# B&R Automation Studio project NAELD004C00R10L518F00 (part 11)

#### Act_OptP0921RstMnl.st
```iecst
ACTION Act_OptP0921RstMnl:

	IF EDGEPOS((bManualMod = FALSE) OR (p_eInShutterStatus = Error) OR (p_eInShutterStatus2 = Error) OR (p_eInShutterStatus3 = Error)) THEN

		eInShutterAct	:= PneuActIdle;
		eInShutterAct2	:= PneuActIdle;
		eInShutterAct3	:= PneuActIdle;

		tyP0921InletNOutletShutter.tyInletShutterDC.tyBtnClose.bRtCompl	:= FALSE;
		tyP0921InletNOutletShutter.tyInletShutterDC.tyBtnClose.bValue	:= FALSE;
		tyP0921InletNOutletShutter.tyInletShutterDC.tyBtnOpen.bRtCompl	:= FALSE;
		tyP0921InletNOutletShutter.tyInletShutterDC.tyBtnOpen.bValue	:= TRUE;

		tyP0921InletNOutletShutter.tyInletShutterFB.tyBtnClose.bRtCompl	:= FALSE;
		tyP0921InletNOutletShutter.tyInletShutterFB.tyBtnClose.bValue	:= FALSE;
		tyP0921InletNOutletShutter.tyInletShutterFB.tyBtnOpen.bRtCompl	:= FALSE;
		tyP0921InletNOutletShutter.tyInletShutterFB.tyBtnOpen.bValue	:= FALSE;

		//in shutt 2
		tyP0921InletNOutletShutter.tyInletShutterDC2.tyBtnClose.bRtCompl	:= FALSE;
		tyP0921InletNOutletShutter.tyInletShutterDC2.tyBtnClose.bValue	:= FALSE;
		tyP0921InletNOutletShutter.tyInletShutterDC2.tyBtnOpen.bRtCompl	:= FALSE;
		tyP0921InletNOutletShutter.tyInletShutterDC2.tyBtnOpen.bValue	:= TRUE;

		tyP0921InletNOutletShutter.tyInletShutterFB2.tyBtnClose.bRtCompl	:= FALSE;
		tyP0921InletNOutletShutter.tyInletShutterFB2.tyBtnClose.bValue	:= FALSE;
		tyP0921InletNOutletShutter.tyInletShutterFB2.tyBtnOpen.bRtCompl	:= FALSE;
		tyP0921InletNOutletShutter.tyInletShutterFB2.tyBtnOpen.bValue	:= FALSE;

		//in shutt3
		tyP0921InletNOutletShutter.tyInletShutterDC3.tyBtnClose.bRtCompl	:= FALSE;
		tyP0921InletNOutletShutter.tyInletShutterDC3.tyBtnClose.bValue	:= FALSE;
		tyP0921InletNOutletShutter.tyInletShutterDC3.tyBtnOpen.bRtCompl	:= FALSE;
		tyP0921InletNOutletShutter.tyInletShutterDC3.tyBtnOpen.bValue	:= TRUE;

		tyP0921InletNOutletShutter.tyInletShutterFB3.tyBtnClose.bRtCompl	:= FALSE;
		tyP0921InletNOutletShutter.tyInletShutterFB3.tyBtnClose.bValue	:= FALSE;
		tyP0921InletNOutletShutter.tyInletShutterFB3.tyBtnOpen.bRtCompl	:= FALSE;
		tyP0921InletNOutletShutter.tyInletShutterFB3.tyBtnOpen.bValue	:= FALSE;

	END_IF

	IF EDGEPOS((bManualMod = FALSE) OR (p_eOutShutterStatus = Error) OR (p_eOutShutterStatus2 = Error) ) THEN

		eOutShutterAct	:= PneuActIdle;
		eOutShutterAct2	:= PneuActIdle;

		tyP0921InletNOutletShutter.tyOutletShutterDC.tyBtnClose.bRtCompl	:= FALSE;
		tyP0921InletNOutletShutter.tyOutletShutterDC.tyBtnClose.bValue		:= FALSE;
		tyP0921InletNOutletShutter.tyOutletShutterDC.tyBtnOpen.bRtCompl		:= FALSE;
		tyP0921InletNOutletShutter.tyOutletShutterDC.tyBtnOpen.bValue		:= FALSE;

		tyP0921InletNOutletShutter.tyOutletShutterFB.tyBtnClose.bRtCompl	:= FALSE;
		tyP0921InletNOutletShutter.tyOutletShutterFB.tyBtnClose.bValue		:= FALSE;
		tyP0921InletNOutletShutter.tyOutletShutterFB.tyBtnOpen.bRtCompl		:= FALSE;
		tyP0921InletNOutletShutter.tyOutletShutterFB.tyBtnOpen.bValue		:= FALSE;

		tyP0921InletNOutletShutter.tyOutletShutterDC2.tyBtnClose.bRtCompl	:= FALSE;
		tyP0921InletNOutletShutter.tyOutletShutterDC2.tyBtnClose.bValue		:= FALSE;
		tyP0921InletNOutletShutter.tyOutletShutterDC2.tyBtnOpen.bRtCompl	:= FALSE;
		tyP0921InletNOutletShutter.tyOutletShutterDC2.tyBtnOpen.bValue		:= FALSE;

		tyP0921InletNOutletShutter.tyOutletShutterFB2.tyBtnClose.bRtCompl	:= FALSE;
		tyP0921InletNOutletShutter.tyOutletShutterFB2.tyBtnClose.bValue		:= FALSE;
		tyP0921InletNOutletShutter.tyOutletShutterFB2.tyBtnOpen.bRtCompl	:= FALSE;
		tyP0921InletNOutletShutter.tyOutletShutterFB2.tyBtnOpen.bValue		:= FALSE;

	END_IF

	IF EDGEPOS(bManualMod = FALSE) THEN

		//In Shutter
		tyP0921InletNOutletShutter.tyInletShutterCom.tyBtnSwitch.bValue		:= FALSE;
		tyP0921InletNOutletShutter.tyInletShutterCom2.tyBtnSwitch.bValue		:= FALSE;

		fUIInRtStatHide(ADR(tyP0921InletNOutletShutter.tyInletShutterDC.tyLyr.uiRtStat));
		fUIInRtStatOff(ADR(tyP0921InletNOutletShutter.tyInletShutterFB.tyLyr.uiRtStat));

		//Out Shutter
		tyP0921InletNOutletShutter.tyOutletShutterCom.tyBtnSwitch.bValue   := FALSE;
		tyP0921InletNOutletShutter.tyOutletShutterCom2.tyBtnSwitch.bValue   := FALSE;

		fUIInRtStatHide(ADR(tyP0921InletNOutletShutter.tyOutletShutterDC.tyLyr.uiRtStat));
		fUIInRtStatOff(ADR(tyP0921InletNOutletShutter.tyOutletShutterFB.tyLyr.uiRtStat));

	END_IF

END_ACTION
```

#### Act_OptP0921InletShutterChgLyr2.st
```iecst
ACTION Act_OptP0921InletShutterChgLyr2:

//	tyP0921InletNOutletShutter.tyInletShutterFB.tyLyr.uiRtStat.0	:= NOT(p_tyNtParamCurr.bProjInletShutPrep);

	IF p_tyNtParamCurr.bProjInletShutPrep THEN
		IF tyP0921InletNOutletShutter.tyInletShutterCom2.tyBtnSwitch.bRtCompl THEN
			tyP0921InletNOutletShutter.tyInletShutterCom2.tyBtnSwitch.bRtCompl := FALSE;

			IF tyP0921InletNOutletShutter.tyInletShutterCom2.tyBtnSwitch.bValue = TRUE THEN
				fUIInRtStatOff(ADR(tyP0921InletNOutletShutter.tyInletShutterDC2.tyLyr.uiRtStat));
				fUIInRtStatHide(ADR(tyP0921InletNOutletShutter.tyInletShutterFB2.tyLyr.uiRtStat));
			ELSE
				fUIInRtStatHide(ADR(tyP0921InletNOutletShutter.tyInletShutterDC2.tyLyr.uiRtStat));
				fUIInRtStatOff(ADR(tyP0921InletNOutletShutter.tyInletShutterFB2.tyLyr.uiRtStat));
			END_IF

		END_IF
	ELSE
		fUIInRtStatHide(ADR(tyP0921InletNOutletShutter.tyInletShutterDC2.tyLyr.uiRtStat));
		fUIInRtStatHide(ADR(tyP0921InletNOutletShutter.tyInletShutterFB2.tyLyr.uiRtStat));

	END_IF

END_ACTION
```

#### Act_OptP0921InletShutterSen2.st
```iecst
ACTION Act_OptP0921InletShutterSen2:

	tyP0921InletNOutletShutter.tyInletShutterCom2.tyBtnOpenRS.bValue		:= p_tyDI.bInShutterOpenRS2;
	tyP0921InletNOutletShutter.tyInletShutterCom2.tyBtnCloseRS.bValue	:= p_tyDI.bInShutterCloseRS2;

	//Machine Bitmap ,13close 14open
	IF   (p_tyNtParamCurr.eProjMag = LDMagDual AND p_tyNtParamCurr.bMagAutoVerifyPrep = FALSE)
		OR (p_tyNtParamCurr.eProjMag = LDMagTriple AND p_tyNtParamCurr.bMagAutoVerifyPrep = FALSE)
		OR (p_tyNtParamCurr.eProjMag = LDMagDual AND p_tyNtParamCurr.bMagAutoVerifyPrep = TRUE)
		THEN
		IF p_tyDI.bInShutterOpenRS2 = TRUE THEN
			tyP0921InletNOutletShutter.tyInletShutterCom2.tyBitmapMc.uiValueIdx	:= 2;
		ELSIF p_tyNtParamCurr.bProjCurtainSenPrep THEN
			tyP0921InletNOutletShutter.tyInletShutterCom2.tyBitmapMc.uiValueIdx	:= 0+4; //16
		ELSE
			tyP0921InletNOutletShutter.tyInletShutterCom2.tyBitmapMc.uiValueIdx	:= 0;
		END_IF
	ELSIF p_tyNtParamCurr.eProjMag = LDMagTriple AND p_tyNtParamCurr.bMagAutoVerifyPrep = TRUE
		THEN
		IF p_tyDI.bInShutterOpenRS2 = TRUE THEN
			tyP0921InletNOutletShutter.tyInletShutterCom2.tyBitmapMc.uiValueIdx	:= 28;
		ELSE
			tyP0921InletNOutletShutter.tyInletShutterCom2.tyBitmapMc.uiValueIdx	:= 27;
		END_IF

	ELSIF p_tyNtParamCurr.eProjMag = LDMagQuadruple AND p_tyNtParamCurr.bMagAutoVerifyPrep = TRUE
		THEN
		IF p_tyDI.bInShutterOpenRS2 = TRUE THEN
			tyP0921InletNOutletShutter.tyInletShutterCom2.tyBitmapMc.uiValueIdx	:= 51;
		ELSE
			tyP0921InletNOutletShutter.tyInletShutterCom2.tyBitmapMc.uiValueIdx	:= 50;
		END_IF
	END_IF

	IF p_tyNtParamCurr.eProjMag = LDMagTriple AND p_tyNtParamCurr.bProjLifterMagPlatform THEN
		IF 	tyP0921InletNOutletShutter.tyInletShutterCom2.tyBitmapMc.uiValueIdx < 400 THEN
			tyP0921InletNOutletShutter.tyInletShutterCom2.tyBitmapMc.uiValueIdx	:= tyP0921InletNOutletShutter.tyInletShutterCom2.tyBitmapMc.uiValueIdx + 400;
		END_IF
	ELSIF p_tyNtParamCurr.eProjMag = LDMagTriple AND p_tyNtParamCurr.bMagAutoVerifyPrep = FALSE AND p_tyNtParamCurr.bProjMotorizedPullerPrep = FALSE
		THEN
		IF 	tyP0921InletNOutletShutter.tyInletShutterCom2.tyBitmapMc.uiValueIdx < 100 THEN
			tyP0921InletNOutletShutter.tyInletShutterCom2.tyBitmapMc.uiValueIdx	:= tyP0921InletNOutletShutter.tyInletShutterCom2.tyBitmapMc.uiValueIdx + 100;
		END_IF
	ELSIF p_tyNtParamCurr.eProjMag = LDMagTriple AND p_tyNtParamCurr.bMagAutoVerifyPrep = FALSE AND p_tyNtParamCurr.bProjMotorizedPullerPrep
		AND p_tyNtParamCurr.bProjCurtainSenPrep THEN //curtain
		IF 	tyP0921InletNOutletShutter.tyInletShutterCom2.tyBitmapMc.uiValueIdx < 375-13-1 THEN
			tyP0921InletNOutletShutter.tyInletShutterCom2.tyBitmapMc.uiValueIdx	:= tyP0921InletNOutletShutter.tyInletShutterCom2.tyBitmapMc.uiValueIdx + 375-13-1;
		END_IF
	ELSIF (p_tyNtParamCurr.eProjMag = LDMagDual OR p_tyNtParamCurr.eProjMag = LDMagTriple)
		AND p_tyNtParamCurr.bMagAutoVerifyPrep = TRUE
		THEN
		IF 	tyP0921InletNOutletShutter.tyInletShutterCom2.tyBitmapMc.uiValueIdx < 200 THEN
			tyP0921InletNOutletShutter.tyInletShutterCom2.tyBitmapMc.uiValueIdx	:= tyP0921InletNOutletShutter.tyInletShutterCom2.tyBitmapMc.uiValueIdx + 200;
		END_IF
	ELSIF (p_tyNtParamCurr.eProjMag = LDMagDual OR p_tyNtParamCurr.eProjMag = LDMagTriple) AND p_tyNtParamCurr.bMagAutoVerifyPrep = FALSE AND  p_tyNtParamCurr.bProjMotorizedPullerPrep = FALSE THEN
		IF 	tyP0921InletNOutletShutter.tyInletShutterCom2.tyBitmapMc.uiValueIdx < 200 THEN
			IF p_tyNtParamCurr.bProjLifterMagPlatform THEN
				tyP0921InletNOutletShutter.tyInletShutterCom2.tyBitmapMc.uiValueIdx	:= tyP0921InletNOutletShutter.tyInletShutterCom2.tyBitmapMc.uiValueIdx + 247;
			ELSE
				tyP0921InletNOutletShutter.tyInletShutterCom2.tyBitmapMc.uiValueIdx	:= tyP0921InletNOutletShutter.tyInletShutterCom2.tyBitmapMc.uiValueIdx + 200;
			END_IF
		END_IF
	ELSIF (p_tyNtParamCurr.eProjMag = LDMagDual OR p_tyNtParamCurr.eProjMag = LDMagTriple) AND p_tyNtParamCurr.bMagAutoVerifyPrep = FALSE AND p_tyNtParamCurr.bProjMotorizedPullerPrep = TRUE
		THEN
		IF 	tyP0921InletNOutletShutter.tyInletShutterCom2.tyBitmapMc.uiValueIdx < 300 THEN
			tyP0921InletNOutletShutter.tyInletShutterCom2.tyBitmapMc.uiValueIdx	:= tyP0921InletNOutletShutter.tyInletShutterCom2.tyBitmapMc.uiValueIdx + 300;
		END_IF
	END_IF
END_ACTION
```

#### Act_OptP0921InletShutterFB2.st
```iecst
ACTION Act_OptP0921InletShutterFB2:

	IF tyP0921InletNOutletShutter.tyInletShutterCom2.tyBtnSwitch.bValue = FALSE THEN

		IF tyP0921InletNOutletShutter.tyInletShutterFB2.tyBtnOpen.bRtCompl = TRUE THEN
			tyP0921InletNOutletShutter.tyInletShutterFB2.tyBtnOpen.bRtCompl	:= FALSE;

			tyP0921InletNOutletShutter.tyInletShutterFB2.tyBtnOpen.bValue	:= TRUE;
			tyP0921InletNOutletShutter.tyInletShutterFB2.tyBtnClose.bValue	:= FALSE;

		ELSIF tyP0921InletNOutletShutter.tyInletShutterFB2.tyBtnClose.bRtCompl = TRUE THEN
			tyP0921InletNOutletShutter.tyInletShutterFB2.tyBtnClose.bRtCompl	:= FALSE;

			tyP0921InletNOutletShutter.tyInletShutterFB2.tyBtnClose.bValue	:= TRUE;
			tyP0921InletNOutletShutter.tyInletShutterFB2.tyBtnOpen.bValue	:= FALSE;
		END_IF

		IF tyP0921InletNOutletShutter.tyInletShutterFB2.tyBtnOpen.bValue = TRUE THEN
			eInShutterAct2	:= PneuActRet;

			IF p_eInShutterStat2 = PneuActRet AND p_eInShutterStatus2 = Done THEN
				eInShutterAct2	:= PneuActIdle;

				tyP0921InletNOutletShutter.tyInletShutterFB2.tyBtnOpen.bValue	:= FALSE;
			ELSIF p_eInShutterStatus2 = Error THEN
				tyP0921InletNOutletShutter.tyInletShutterFB2.tyBtnOpen.bValue	:= FALSE;
			END_IF

		ELSIF tyP0921InletNOutletShutter.tyInletShutterFB2.tyBtnClose.bValue = TRUE THEN
			eInShutterAct2	:= PneuActExt;

			IF p_eInShutterStat2 = PneuActExt AND p_eInShutterStatus2 = Done THEN
				eInShutterAct2	:= PneuActIdle;

				tyP0921InletNOutletShutter.tyInletShutterFB2.tyBtnClose.bValue := FALSE;
			ELSIF p_eInShutterStatus2 = Error THEN
				tyP0921InletNOutletShutter.tyInletShutterFB2.tyBtnClose.bValue := FALSE;
			END_IF
		END_IF

		//Update Direct Control Status
		tyP0921InletNOutletShutter.tyInletShutterDC2.tyBtnOpen.bRtCompl	:= FALSE;
		tyP0921InletNOutletShutter.tyInletShutterDC2.tyBtnClose.bRtCompl	:= FALSE;
		tyP0921InletNOutletShutter.tyInletShutterDC2.tyBtnOpen.bValue	:= p_bInShutterRetCtrl2;
		tyP0921InletNOutletShutter.tyInletShutterDC2.tyBtnClose.bValue	:= p_bInShutterExtCtrl2;

	END_IF

END_ACTION
```

#### Act_OptP0921InletShutterFBStat2.st
```iecst
ACTION Act_OptP0921InletShutterFBStat2:

	tyP0921InletNOutletShutter.tyInletShutterFB2.tyStringStat.sValue	:= p_sInShutterStatTxt2;

END_ACTION
```

#### Act_OptP0921InletShutterDC2.st
```iecst
ACTION Act_OptP0921InletShutterDC2:

	IF tyP0921InletNOutletShutter.tyInletShutterCom2.tyBtnSwitch.bValue = TRUE THEN
		IF p_bInShutterTwoCtrlOut2 = FALSE THEN
			IF tyP0921InletNOutletShutter.tyInletShutterDC2.tyBtnOpen.bRtCompl = TRUE THEN
				tyP0921InletNOutletShutter.tyInletShutterDC2.tyBtnOpen.bValue	:= TRUE;
				tyP0921InletNOutletShutter.tyInletShutterDC2.tyBtnClose.bValue	:= FALSE;

				eInShutterAct2	:= PneuActSetRet;

				IF p_eInShutterStat2 = PneuActSetRet AND p_eInShutterStatus2 = Done THEN
					eInShutterAct2	:= PneuActIdle;

					tyP0921InletNOutletShutter.tyInletShutterDC2.tyBtnOpen.bRtCompl	:= FALSE;
				END_IF

			ELSIF tyP0921InletNOutletShutter.tyInletShutterDC2.tyBtnClose.bRtCompl = TRUE THEN
				tyP0921InletNOutletShutter.tyInletShutterDC2.tyBtnClose.bValue	:= TRUE;
				tyP0921InletNOutletShutter.tyInletShutterDC2.tyBtnOpen.bValue	:= FALSE;

				eInShutterAct2	:= PneuActSetExt;

				IF p_eInShutterStat2 = PneuActSetExt AND p_eInShutterStatus2 = Done THEN
					eInShutterAct2	:= PneuActIdle;

					tyP0921InletNOutletShutter.tyInletShutterDC2.tyBtnClose.bRtCompl	:= FALSE;
				END_IF
			END_IF

		ELSE
			IF (tyP0921InletNOutletShutter.tyInletShutterDC2.tyBtnOpen.bRtCompl = TRUE) OR (tyP0921InletNOutletShutter.tyInletShutterDC2.tyBtnClose.bRtCompl = TRUE) THEN
				IF (tyP0921InletNOutletShutter.tyInletShutterDC2.tyBtnOpen.bValue = TRUE) AND (tyP0921InletNOutletShutter.tyInletShutterDC2.tyBtnClose.bValue = TRUE) THEN
					eInShutterAct2	:= PneuActSetAll;

					IF p_eInShutterStat2 = PneuActSetAll AND p_eInShutterStatus2 = Done THEN
						eInShutterAct2	:= PneuActIdle;

						tyP0921InletNOutletShutter.tyInletShutterDC2.tyBtnOpen.bRtCompl	:= FALSE;
						tyP0921InletNOutletShutter.tyInletShutterDC2.tyBtnClose.bRtCompl	:= FALSE;
					END_IF

				ELSIF (tyP0921InletNOutletShutter.tyInletShutterDC2.tyBtnOpen.bValue = TRUE) AND (tyP0921InletNOutletShutter.tyInletShutterDC2.tyBtnClose.bValue = FALSE) THEN
					eInShutterAct2	:= PneuActSetRet;

					IF p_eInShutterStat2 = PneuActSetRet AND p_eInShutterStatus2 = Done THEN
						eInShutterAct2	:= PneuActIdle;

						tyP0921InletNOutletShutter.tyInletShutterDC2.tyBtnOpen.bRtCompl	:= FALSE;
						tyP0921InletNOutletShutter.tyInletShutterDC2.tyBtnClose.bRtCompl	:= FALSE;
					END_IF

				ELSIF (tyP0921InletNOutletShutter.tyInletShutterDC2.tyBtnOpen.bValue = FALSE) AND (tyP0921InletNOutletShutter.tyInletShutterDC2.tyBtnClose.bValue = TRUE) THEN
					eInShutterAct2	:= PneuActSetExt;

					IF p_eInShutterStat2 = PneuActSetExt AND p_eInShutterStatus2 = Done THEN
						eInShutterAct2	:= PneuActIdle;

						tyP0921InletNOutletShutter.tyInletShutterDC2.tyBtnOpen.bRtCompl	:= FALSE;
						tyP0921InletNOutletShutter.tyInletShutterDC2.tyBtnClose.bRtCompl	:= FALSE;
					END_IF

				ELSE
					eInShutterAct2	:= PneuActRstAll;

					IF p_eInShutterStat2 = PneuActRstAll AND p_eInShutterStatus2 = Done THEN
						eInShutterAct2	:= PneuActIdle;

						tyP0921InletNOutletShutter.tyInletShutterDC2.tyBtnOpen.bRtCompl	:= FALSE;
						tyP0921InletNOutletShutter.tyInletShutterDC2.tyBtnClose.bRtCompl	:= FALSE;
					END_IF

				END_IF
			END_IF
		END_IF

		tyP0921InletNOutletShutter.tyInletShutterFB2.tyBtnClose.bRtCompl	:= FALSE;
		tyP0921InletNOutletShutter.tyInletShutterFB2.tyBtnClose.bValue	:= FALSE;
		tyP0921InletNOutletShutter.tyInletShutterFB2.tyBtnOpen.bRtCompl	:= FALSE;
		tyP0921InletNOutletShutter.tyInletShutterFB2.tyBtnOpen.bValue	:= FALSE;

	END_IF

END_ACTION
```

#### Act_OptP0921InletShutterChgLyr3.st
```iecst
ACTION Act_OptP0921InletShutterChgLyr3:

//	tyP0921InletNOutletShutter.tyInletShutterFB2.tyLyr.uiRtStat.0	:= NOT(p_tyNtParamCurr.bProjInletShutPrep);

	IF p_tyNtParamCurr.bProjInletShutPrep THEN
		IF tyP0921InletNOutletShutter.tyInletShutterCom3.tyBtnSwitch.bRtCompl THEN
			tyP0921InletNOutletShutter.tyInletShutterCom3.tyBtnSwitch.bRtCompl := FALSE;

			IF tyP0921InletNOutletShutter.tyInletShutterCom3.tyBtnSwitch.bValue = TRUE THEN
				fUIInRtStatOff(ADR(tyP0921InletNOutletShutter.tyInletShutterDC3.tyLyr.uiRtStat));
				fUIInRtStatHide(ADR(tyP0921InletNOutletShutter.tyInletShutterFB3.tyLyr.uiRtStat));
			ELSE
				fUIInRtStatHide(ADR(tyP0921InletNOutletShutter.tyInletShutterDC3.tyLyr.uiRtStat));
				fUIInRtStatOff(ADR(tyP0921InletNOutletShutter.tyInletShutterFB3.tyLyr.uiRtStat));
			END_IF

		END_IF
	ELSE
		fUIInRtStatHide(ADR(tyP0921InletNOutletShutter.tyInletShutterDC3.tyLyr.uiRtStat));
		fUIInRtStatHide(ADR(tyP0921InletNOutletShutter.tyInletShutterFB3.tyLyr.uiRtStat));

	END_IF

END_ACTION
```

#### Act_OptP0921InletShutterSen3.st
```iecst
ACTION Act_OptP0921InletShutterSen3:

	tyP0921InletNOutletShutter.tyInletShutterCom3.tyBtnOpenRS.bValue		:= p_tyDI.bInShutterOpenRS3;
	tyP0921InletNOutletShutter.tyInletShutterCom3.tyBtnCloseRS.bValue	:= p_tyDI.bInShutterCloseRS3;

	//Machine Bitmap, 15close ,16open
	IF   (p_tyNtParamCurr.eProjMag = LDMagDual AND p_tyNtParamCurr.bMagAutoVerifyPrep = FALSE)
		OR (p_tyNtParamCurr.eProjMag = LDMagTriple AND p_tyNtParamCurr.bMagAutoVerifyPrep = FALSE)
		OR (p_tyNtParamCurr.eProjMag = LDMagDual AND p_tyNtParamCurr.bMagAutoVerifyPrep = TRUE)
		THEN
		IF p_tyDI.bInShutterOpenRS3 = TRUE THEN
			tyP0921InletNOutletShutter.tyInletShutterCom3.tyBitmapMc.uiValueIdx	:= 3;
		ELSIF p_tyNtParamCurr.bProjCurtainSenPrep THEN
			tyP0921InletNOutletShutter.tyInletShutterCom3.tyBitmapMc.uiValueIdx	:= 0+4; //
		ELSE
			tyP0921InletNOutletShutter.tyInletShutterCom3.tyBitmapMc.uiValueIdx	:= 0;
		END_IF
	ELSIF p_tyNtParamCurr.eProjMag = LDMagTriple AND p_tyNtParamCurr.bMagAutoVerifyPrep = TRUE THEN
		IF p_tyDI.bInShutterOpenRS3 = TRUE THEN
			tyP0921InletNOutletShutter.tyInletShutterCom3.tyBitmapMc.uiValueIdx	:= 28;
		ELSE
			tyP0921InletNOutletShutter.tyInletShutterCom3.tyBitmapMc.uiValueIdx	:= 27;
		END_IF

	ELSIF p_tyNtParamCurr.eProjMag = LDMagQuadruple AND p_tyNtParamCurr.bMagAutoVerifyPrep = TRUE THEN
		IF p_tyDI.bInShutterOpenRS3 = TRUE THEN
			tyP0921InletNOutletShutter.tyInletShutterCom3.tyBitmapMc.uiValueIdx	:= 51;
		ELSE
			tyP0921InletNOutletShutter.tyInletShutterCom3.tyBitmapMc.uiValueIdx	:= 50;
		END_IF
	END_IF

	IF p_tyNtParamCurr.eProjMag = LDMagTriple AND p_tyNtParamCurr.bProjLifterMagPlatform THEN
		IF 	tyP0921InletNOutletShutter.tyInletShutterCom3.tyBitmapMc.uiValueIdx < 400 THEN
			tyP0921InletNOutletShutter.tyInletShutterCom3.tyBitmapMc.uiValueIdx	:= tyP0921InletNOutletShutter.tyInletShutterCom3.tyBitmapMc.uiValueIdx + 400;
		END_IF
	ELSIF p_tyNtParamCurr.eProjMag = LDMagTriple AND p_tyNtParamCurr.bMagAutoVerifyPrep = FALSE AND p_tyNtParamCurr.bProjMotorizedPullerPrep = FALSE
		THEN
		IF 	tyP0921InletNOutletShutter.tyInletShutterCom3.tyBitmapMc.uiValueIdx < 100 THEN
			tyP0921InletNOutletShutter.tyInletShutterCom3.tyBitmapMc.uiValueIdx	:= tyP0921InletNOutletShutter.tyInletShutterCom3.tyBitmapMc.uiValueIdx + 100;
		END_IF
	ELSIF p_tyNtParamCurr.eProjMag = LDMagTriple AND p_tyNtParamCurr.bMagAutoVerifyPrep = FALSE AND p_tyNtParamCurr.bProjMotorizedPullerPrep
		AND p_tyNtParamCurr.bProjCurtainSenPrep THEN
		IF 	tyP0921InletNOutletShutter.tyInletShutterCom3.tyBitmapMc.uiValueIdx < 377-15-3 THEN
			tyP0921InletNOutletShutter.tyInletShutterCom3.tyBitmapMc.uiValueIdx	:= tyP0921InletNOutletShutter.tyInletShutterCom3.tyBitmapMc.uiValueIdx + 377-15-3;//3open
		END_IF
	ELSIF (p_tyNtParamCurr.eProjMag = LDMagDual OR p_tyNtParamCurr.eProjMag = LDMagTriple)
		AND p_tyNtParamCurr.bMagAutoVerifyPrep = TRUE
		THEN
		IF 	tyP0921InletNOutletShutter.tyInletShutterCom3.tyBitmapMc.uiValueIdx < 200 THEN
			tyP0921InletNOutletShutter.tyInletShutterCom3.tyBitmapMc.uiValueIdx	:= tyP0921InletNOutletShutter.tyInletShutterCom3.tyBitmapMc.uiValueIdx + 200;
		END_IF
	ELSIF (p_tyNtParamCurr.eProjMag = LDMagDual OR p_tyNtParamCurr.eProjMag = LDMagTriple) AND p_tyNtParamCurr.bMagAutoVerifyPrep = FALSE AND  p_tyNtParamCurr.bProjMotorizedPullerPrep = FALSE THEN
		IF 	tyP0921InletNOutletShutter.tyInletShutterCom3.tyBitmapMc.uiValueIdx < 200 THEN
			IF p_tyNtParamCurr.bProjLifterMagPlatform THEN
				tyP0921InletNOutletShutter.tyInletShutterCom3.tyBitmapMc.uiValueIdx	:= tyP0921InletNOutletShutter.tyInletShutterCom3.tyBitmapMc.uiValueIdx + 247;
			ELSE
				tyP0921InletNOutletShutter.tyInletShutterCom3.tyBitmapMc.uiValueIdx	:= tyP0921InletNOutletShutter.tyInletShutterCom3.tyBitmapMc.uiValueIdx + 200;
			END_IF
		END_IF
	ELSIF (p_tyNtParamCurr.eProjMag = LDMagDual OR p_tyNtParamCurr.eProjMag = LDMagTriple) AND p_tyNtParamCurr.bMagAutoVerifyPrep = FALSE AND p_tyNtParamCurr.bProjMotorizedPullerPrep = TRUE
		THEN
		IF 	tyP0921InletNOutletShutter.tyInletShutterCom3.tyBitmapMc.uiValueIdx < 300 THEN
			tyP0921InletNOutletShutter.tyInletShutterCom3.tyBitmapMc.uiValueIdx	:= tyP0921InletNOutletShutter.tyInletShutterCom3.tyBitmapMc.uiValueIdx + 300;
		END_IF
	END_IF
END_ACTION
```

#### Act_OptP0921InletShutterFB3.st
```iecst
ACTION Act_OptP0921InletShutterFB3:

	IF tyP0921InletNOutletShutter.tyInletShutterCom3.tyBtnSwitch.bValue = FALSE THEN

		IF tyP0921InletNOutletShutter.tyInletShutterFB3.tyBtnOpen.bRtCompl = TRUE THEN
			tyP0921InletNOutletShutter.tyInletShutterFB3.tyBtnOpen.bRtCompl	:= FALSE;

			tyP0921InletNOutletShutter.tyInletShutterFB3.tyBtnOpen.bValue	:= TRUE;
			tyP0921InletNOutletShutter.tyInletShutterFB3.tyBtnClose.bValue	:= FALSE;

		ELSIF tyP0921InletNOutletShutter.tyInletShutterFB3.tyBtnClose.bRtCompl = TRUE THEN
			tyP0921InletNOutletShutter.tyInletShutterFB3.tyBtnClose.bRtCompl	:= FALSE;

			tyP0921InletNOutletShutter.tyInletShutterFB3.tyBtnClose.bValue	:= TRUE;
			tyP0921InletNOutletShutter.tyInletShutterFB3.tyBtnOpen.bValue	:= FALSE;
		END_IF

		IF tyP0921InletNOutletShutter.tyInletShutterFB3.tyBtnOpen.bValue = TRUE THEN
			eInShutterAct3	:= PneuActRet;

			IF p_eInShutterStat3 = PneuActRet AND p_eInShutterStatus3 = Done THEN
				eInShutterAct3	:= PneuActIdle;

				tyP0921InletNOutletShutter.tyInletShutterFB3.tyBtnOpen.bValue	:= FALSE;
			ELSIF p_eInShutterStatus3 = Error THEN
				tyP0921InletNOutletShutter.tyInletShutterFB3.tyBtnOpen.bValue	:= FALSE;
			END_IF

		ELSIF tyP0921InletNOutletShutter.tyInletShutterFB3.tyBtnClose.bValue = TRUE THEN
			eInShutterAct3	:= PneuActExt;

			IF p_eInShutterStat3 = PneuActExt AND p_eInShutterStatus3 = Done THEN
				eInShutterAct3	:= PneuActIdle;

				tyP0921InletNOutletShutter.tyInletShutterFB3.tyBtnClose.bValue := FALSE;
			ELSIF p_eInShutterStatus3 = Error THEN
				tyP0921InletNOutletShutter.tyInletShutterFB3.tyBtnClose.bValue := FALSE;
			END_IF
		END_IF

		//Update Direct Control Status
		tyP0921InletNOutletShutter.tyInletShutterDC3.tyBtnOpen.bRtCompl	:= FALSE;
		tyP0921InletNOutletShutter.tyInletShutterDC3.tyBtnClose.bRtCompl	:= FALSE;
		tyP0921InletNOutletShutter.tyInletShutterDC3.tyBtnOpen.bValue	:= p_bInShutterRetCtrl3;
		tyP0921InletNOutletShutter.tyInletShutterDC3.tyBtnClose.bValue	:= p_bInShutterExtCtrl3;

	END_IF

END_ACTION
```

#### Act_OptP0921InletShutterFBStat3.st
```iecst
ACTION Act_OptP0921InletShutterFBStat3:

	tyP0921InletNOutletShutter.tyInletShutterFB3.tyStringStat.sValue	:= p_sInShutterStatTxt3;

END_ACTION
```

#### Act_OptP0921InletShutterDC3.st
```iecst
ACTION Act_OptP0921InletShutterDC3:

	IF tyP0921InletNOutletShutter.tyInletShutterCom3.tyBtnSwitch.bValue = TRUE THEN
		IF p_bInShutterTwoCtrlOut = FALSE THEN
			IF tyP0921InletNOutletShutter.tyInletShutterDC3.tyBtnOpen.bRtCompl = TRUE THEN
				tyP0921InletNOutletShutter.tyInletShutterDC3.tyBtnOpen.bValue	:= TRUE;
				tyP0921InletNOutletShutter.tyInletShutterDC3.tyBtnClose.bValue	:= FALSE;

				eInShutterAct3	:= PneuActSetRet;

				IF p_eInShutterStat3 = PneuActSetRet AND p_eInShutterStatus3 = Done THEN
					eInShutterAct3	:= PneuActIdle;

					tyP0921InletNOutletShutter.tyInletShutterDC3.tyBtnOpen.bRtCompl	:= FALSE;
				END_IF

			ELSIF tyP0921InletNOutletShutter.tyInletShutterDC3.tyBtnClose.bRtCompl = TRUE THEN
				tyP0921InletNOutletShutter.tyInletShutterDC3.tyBtnClose.bValue	:= TRUE;
				tyP0921InletNOutletShutter.tyInletShutterDC3.tyBtnOpen.bValue	:= FALSE;

				eInShutterAct3	:= PneuActSetExt;

				IF p_eInShutterStat3 = PneuActSetExt AND p_eInShutterStatus3 = Done THEN
					eInShutterAct3	:= PneuActIdle;

					tyP0921InletNOutletShutter.tyInletShutterDC3.tyBtnClose.bRtCompl	:= FALSE;
				END_IF
			END_IF

		ELSE
			IF (tyP0921InletNOutletShutter.tyInletShutterDC3.tyBtnOpen.bRtCompl = TRUE) OR (tyP0921InletNOutletShutter.tyInletShutterDC3.tyBtnClose.bRtCompl = TRUE) THEN
				IF (tyP0921InletNOutletShutter.tyInletShutterDC3.tyBtnOpen.bValue = TRUE) AND (tyP0921InletNOutletShutter.tyInletShutterDC3.tyBtnClose.bValue = TRUE) THEN
					eInShutterAct3	:= PneuActSetAll;

					IF p_eInShutterStat3 = PneuActSetAll AND p_eInShutterStatus3 = Done THEN
						eInShutterAct3	:= PneuActIdle;

						tyP0921InletNOutletShutter.tyInletShutterDC3.tyBtnOpen.bRtCompl	:= FALSE;
						tyP0921InletNOutletShutter.tyInletShutterDC3.tyBtnClose.bRtCompl	:= FALSE;
					END_IF

				ELSIF (tyP0921InletNOutletShutter.tyInletShutterDC3.tyBtnOpen.bValue = TRUE) AND (tyP0921InletNOutletShutter.tyInletShutterDC3.tyBtnClose.bValue = FALSE) THEN
					eInShutterAct3	:= PneuActSetRet;

					IF p_eInShutterStat3 = PneuActSetRet AND p_eInShutterStatus3 = Done THEN
						eInShutterAct3	:= PneuActIdle;

						tyP0921InletNOutletShutter.tyInletShutterDC3.tyBtnOpen.bRtCompl	:= FALSE;
						tyP0921InletNOutletShutter.tyInletShutterDC3.tyBtnClose.bRtCompl	:= FALSE;
					END_IF

				ELSIF (tyP0921InletNOutletShutter.tyInletShutterDC3.tyBtnOpen2.bValue = TRUE) AND (tyP0921InletNOutletShutter.tyInletShutterDC3.tyBtnClose.bValue = FALSE) THEN
					eInShutterAct2	:= PneuActSetRet;

					IF p_eInShutterStat2 = PneuActSetRet AND p_eInShutterStatus2 = Done THEN
						eInShutterAct2	:= PneuActIdle;

						tyP0921InletNOutletShutter.tyInletShutterDC3.tyBtnOpen2.bRtCompl	:= FALSE;
						tyP0921InletNOutletShutter.tyInletShutterDC3.tyBtnClose.bRtCompl	:= FALSE;
					END_IF

				ELSIF (tyP0921InletNOutletShutter.tyInletShutterDC3.tyBtnOpen3.bValue = TRUE) AND (tyP0921InletNOutletShutter.tyInletShutterDC3.tyBtnClose.bValue = FALSE) THEN
					eInShutterAct3	:= PneuActSetRet;

					IF p_eInShutterStat3 = PneuActSetRet AND p_eInShutterStatus3 = Done THEN
						eInShutterAct3	:= PneuActIdle;

						tyP0921InletNOutletShutter.tyInletShutterDC3.tyBtnOpen3.bRtCompl	:= FALSE;
						tyP0921InletNOutletShutter.tyInletShutterDC3.tyBtnClose.bRtCompl	:= FALSE;
					END_IF

				ELSIF (tyP0921InletNOutletShutter.tyInletShutterDC3.tyBtnOpen.bValue = FALSE) AND (tyP0921InletNOutletShutter.tyInletShutterDC3.tyBtnClose.bValue = TRUE) THEN
					eInShutterAct3	:= PneuActSetExt;

					IF p_eInShutterStat3 = PneuActSetExt AND p_eInShutterStatus3 = Done THEN
						eInShutterAct3	:= PneuActIdle;

						tyP0921InletNOutletShutter.tyInletShutterDC3.tyBtnOpen.bRtCompl	:= FALSE;
						tyP0921InletNOutletShutter.tyInletShutterDC3.tyBtnClose.bRtCompl	:= FALSE;
					END_IF

				ELSE
					eInShutterAct3	:= PneuActRstAll;

					IF p_eInShutterStat3 = PneuActRstAll AND p_eInShutterStatus3 = Done THEN
						eInShutterAct3	:= PneuActIdle;

						tyP0921InletNOutletShutter.tyInletShutterDC3.tyBtnOpen.bRtCompl	:= FALSE;
						tyP0921InletNOutletShutter.tyInletShutterDC3.tyBtnClose.bRtCompl	:= FALSE;
					END_IF

				END_IF
			END_IF
		END_IF

		tyP0921InletNOutletShutter.tyInletShutterFB3.tyBtnClose.bRtCompl	:= FALSE;
		tyP0921InletNOutletShutter.tyInletShutterFB3.tyBtnClose.bValue	:= FALSE;
		tyP0921InletNOutletShutter.tyInletShutterFB3.tyBtnOpen.bRtCompl	:= FALSE;
		tyP0921InletNOutletShutter.tyInletShutterFB3.tyBtnOpen.bValue	:= FALSE;

	END_IF

END_ACTION
```

#### Act_OptP0921OutletShutterChgLyr2.st
```iecst
ACTION Act_OptP0921OutletShutterChgLyr2:

//	tyP0921InletNOutletShutter.tyOutletShutterFB2.tyLyr.uiRtStat.0	:= NOT(p_tyNtParamCurr.bProjOutShutter2Prep);

	IF p_tyNtParamCurr.bProjOutShutter2Prep THEN
		IF	tyP0921InletNOutletShutter.tyOutletShutterCom2.tyBtnSwitch.bRtCompl THEN
				tyP0921InletNOutletShutter.tyOutletShutterCom2.tyBtnSwitch.bRtCompl := FALSE;

			IF tyP0921InletNOutletShutter.tyOutletShutterCom2.tyBtnSwitch.bValue = TRUE THEN
				fUIInRtStatOff(ADR(tyP0921InletNOutletShutter.tyOutletShutterDC2.tyLyr.uiRtStat));
				fUIInRtStatHide(ADR(tyP0921InletNOutletShutter.tyOutletShutterFB2.tyLyr.uiRtStat));
			ELSE
				fUIInRtStatHide(ADR(tyP0921InletNOutletShutter.tyOutletShutterDC2.tyLyr.uiRtStat));
				fUIInRtStatOff(ADR(tyP0921InletNOutletShutter.tyOutletShutterFB2.tyLyr.uiRtStat));
			END_IF

		END_IF
	ELSE
		fUIInRtStatHide(ADR(tyP0921InletNOutletShutter.tyOutletShutterDC2.tyLyr.uiRtStat));
		fUIInRtStatHide(ADR(tyP0921InletNOutletShutter.tyOutletShutterFB2.tyLyr.uiRtStat));

	END_IF

END_ACTION
```

#### Act_OptP0921OutletShutterSen2.st
```iecst
ACTION Act_OptP0921OutletShutterSen2:

	tyP0921InletNOutletShutter.tyOutletShutterCom2.tyBtnOpenRS.bValue	:= p_tyDI.bOutShutterOpenRS2;
	tyP0921InletNOutletShutter.tyOutletShutterCom2.tyBtnCloseRS.bValue	:= p_tyDI.bOutShutterCloseRS2;

	//Machine Bitmap //15open ,16close
	IF   (p_tyNtParamCurr.eProjMag = LDMagDual AND p_tyNtParamCurr.bMagAutoVerifyPrep = FALSE)
		OR (p_tyNtParamCurr.eProjMag = LDMagTriple AND p_tyNtParamCurr.bMagAutoVerifyPrep = FALSE)
		OR (p_tyNtParamCurr.eProjMag = LDMagDual AND p_tyNtParamCurr.bMagAutoVerifyPrep = TRUE)
		THEN
		IF p_tyDI.bOutShutterOpenRS2 = TRUE THEN
			tyP0921InletNOutletShutter.tyOutletShutterCom2.tyBitmapMc.uiValueIdx	:= 1;
		ELSE
			tyP0921InletNOutletShutter.tyOutletShutterCom2.tyBitmapMc.uiValueIdx	:= 0;
		END_IF
	ELSIF p_tyNtParamCurr.eProjMag = LDMagTriple AND p_tyNtParamCurr.bMagAutoVerifyPrep = TRUE
		THEN
		IF p_tyDI.bOutShutterOpenRS2 = TRUE THEN
			tyP0921InletNOutletShutter.tyOutletShutterCom2.tyBitmapMc.uiValueIdx	:= 28;
		ELSE
			tyP0921InletNOutletShutter.tyOutletShutterCom2.tyBitmapMc.uiValueIdx	:= 27;
		END_IF
	ELSIF p_tyNtParamCurr.eProjMag = LDMagQuadruple AND p_tyNtParamCurr.bMagAutoVerifyPrep = TRUE
		THEN
		IF p_tyDI.bOutShutterOpenRS2 = TRUE THEN
			tyP0921InletNOutletShutter.tyOutletShutterCom2.tyBitmapMc.uiValueIdx	:= 51;
		ELSE
			tyP0921InletNOutletShutter.tyOutletShutterCom2.tyBitmapMc.uiValueIdx	:= 50;
		END_IF
	END_IF

	IF p_tyNtParamCurr.eProjMag = LDMagTriple AND p_tyNtParamCurr.bProjLifterMagPlatform THEN //same with bosch curtain
		IF 	tyP0921InletNOutletShutter.tyOutletShutterCom2.tyBitmapMc.uiValueIdx < 400 THEN
			tyP0921InletNOutletShutter.tyOutletShutterCom2.tyBitmapMc.uiValueIdx	:= tyP0921InletNOutletShutter.tyOutletShutterCom2.tyBitmapMc.uiValueIdx + 400;
		END_IF
	ELSIF p_tyNtParamCurr.eProjMag = LDMagTriple AND p_tyNtParamCurr.bMagAutoVerifyPrep = FALSE AND p_tyNtParamCurr.bProjMotorizedPullerPrep = FALSE
		THEN
		IF 	tyP0921InletNOutletShutter.tyOutletShutterCom2.tyBitmapMc.uiValueIdx < 100 THEN
			tyP0921InletNOutletShutter.tyOutletShutterCom2.tyBitmapMc.uiValueIdx	:= tyP0921InletNOutletShutter.tyOutletShutterCom2.tyBitmapMc.uiValueIdx + 100;
		END_IF
	ELSIF p_tyNtParamCurr.eProjMag = LDMagTriple AND p_tyNtParamCurr.bMagAutoVerifyPrep = FALSE AND p_tyNtParamCurr.bProjMotorizedPullerPrep = TRUE
		AND p_tyNtParamCurr.bProjCurtainSenPrep THEN //curtain
		IF 	tyP0921InletNOutletShutter.tyOutletShutterCom2.tyBitmapMc.uiValueIdx < 387-15 THEN
			tyP0921InletNOutletShutter.tyOutletShutterCom2.tyBitmapMc.uiValueIdx	:= tyP0921InletNOutletShutter.tyOutletShutterCom2.tyBitmapMc.uiValueIdx + 387-15;
		END_IF
	ELSIF (p_tyNtParamCurr.eProjMag = LDMagDual OR p_tyNtParamCurr.eProjMag = LDMagTriple)
		AND p_tyNtParamCurr.bMagAutoVerifyPrep = TRUE
		THEN
		IF 	tyP0921InletNOutletShutter.tyOutletShutterCom2.tyBitmapMc.uiValueIdx < 200 THEN
			tyP0921InletNOutletShutter.tyOutletShutterCom2.tyBitmapMc.uiValueIdx	:= tyP0921InletNOutletShutter.tyOutletShutterCom2.tyBitmapMc.uiValueIdx + 200;
		END_IF
	ELSIF (p_tyNtParamCurr.eProjMag = LDMagDual OR p_tyNtParamCurr.eProjMag = LDMagTriple)
		AND p_tyNtParamCurr.bMagAutoVerifyPrep = FALSE  AND p_tyNtParamCurr.bProjMotorizedPullerPrep = TRUE
		THEN
		IF 	tyP0921InletNOutletShutter.tyOutletShutterCom2.tyBitmapMc.uiValueIdx < 300 THEN
			tyP0921InletNOutletShutter.tyOutletShutterCom2.tyBitmapMc.uiValueIdx	:= tyP0921InletNOutletShutter.tyOutletShutterCom2.tyBitmapMc.uiValueIdx + 300;
		END_IF
	ELSIF (p_tyNtParamCurr.eProjMag = LDMagDual OR p_tyNtParamCurr.eProjMag = LDMagTriple)
		AND p_tyNtParamCurr.bMagAutoVerifyPrep = FALSE  AND p_tyNtParamCurr.bProjMotorizedPullerPrep = FALSE
		THEN
		IF 	tyP0921InletNOutletShutter.tyOutletShutterCom2.tyBitmapMc.uiValueIdx < 200 THEN
			IF p_tyNtParamCurr.bProjLifterMagPlatform THEN
				tyP0921InletNOutletShutter.tyOutletShutterCom2.tyBitmapMc.uiValueIdx	:= tyP0921InletNOutletShutter.tyOutletShutterCom2.tyBitmapMc.uiValueIdx + 247;
			ELSE
				IF p_tyNtParamCurr.sJobNo = '2023-0276A01' THEN
					tyP0921InletNOutletShutter.tyOutletShutterCom2.tyBitmapMc.uiValueIdx	:= tyP0921InletNOutletShutter.tyOutletShutterCom2.tyBitmapMc.uiValueIdx + 484-15+2;
				ELSE
					tyP0921InletNOutletShutter.tyOutletShutterCom2.tyBitmapMc.uiValueIdx	:= tyP0921InletNOutletShutter.tyOutletShutterCom2.tyBitmapMc.uiValueIdx + 200;
				END_IF
			END_IF
		END_IF
	END_IF
	END_ACTION
```

#### Act_OptP0921OutletShutterFB2.st
```iecst
ACTION Act_OptP0921OutletShutterFB2:

	IF tyP0921InletNOutletShutter.tyOutletShutterCom2.tyBtnSwitch.bValue = FALSE THEN
		// FB Control
		IF tyP0921InletNOutletShutter.tyOutletShutterFB2.tyBtnOpen.bRtCompl = TRUE THEN
			tyP0921InletNOutletShutter.tyOutletShutterFB2.tyBtnOpen.bRtCompl	:= FALSE;

			tyP0921InletNOutletShutter.tyOutletShutterFB2.tyBtnOpen.bValue	:= TRUE;
			tyP0921InletNOutletShutter.tyOutletShutterFB2.tyBtnClose.bValue	:= FALSE;

		ELSIF tyP0921InletNOutletShutter.tyOutletShutterFB2.tyBtnClose.bRtCompl = TRUE THEN
			tyP0921InletNOutletShutter.tyOutletShutterFB2.tyBtnClose.bRtCompl	:= FALSE;

			tyP0921InletNOutletShutter.tyOutletShutterFB2.tyBtnClose.bValue	:= TRUE;
			tyP0921InletNOutletShutter.tyOutletShutterFB2.tyBtnOpen.bValue	:= FALSE;
		END_IF

		IF tyP0921InletNOutletShutter.tyOutletShutterFB2.tyBtnOpen.bValue = TRUE THEN
			eOutShutterAct2	:= PneuActRet;

			IF p_eOutShutterStat2 = PneuActRet AND p_eOutShutterStatus2 = Done THEN
				eOutShutterAct2	:= PneuActIdle;

				tyP0921InletNOutletShutter.tyOutletShutterFB2.tyBtnOpen.bValue	:= FALSE;
			ELSIF p_eOutShutterStatus2 = Error THEN
				tyP0921InletNOutletShutter.tyOutletShutterFB2.tyBtnOpen.bValue	:= FALSE;
			END_IF

		ELSIF tyP0921InletNOutletShutter.tyOutletShutterFB2.tyBtnClose.bValue = TRUE THEN
			eOutShutterAct2	:= PneuActExt;

			IF p_eOutShutterStat2 = PneuActExt AND p_eOutShutterStatus2 = Done THEN
				eOutShutterAct2	:= PneuActIdle;

				tyP0921InletNOutletShutter.tyOutletShutterFB2.tyBtnClose.bValue := FALSE;
			ELSIF p_eOutShutterStatus2 = Error THEN
				tyP0921InletNOutletShutter.tyOutletShutterFB2.tyBtnClose.bValue := FALSE;
			END_IF
		END_IF

		//UpdateStatus
		tyP0921InletNOutletShutter.tyOutletShutterDC2.tyBtnClose.bRtCompl	:= FALSE;
		tyP0921InletNOutletShutter.tyOutletShutterDC2.tyBtnOpen.bRtCompl		:= FALSE;
		tyP0921InletNOutletShutter.tyOutletShutterDC2.tyBtnClose.bValue		:= p_bOutShutterExtCtrl2;
		tyP0921InletNOutletShutter.tyOutletShutterDC2.tyBtnOpen.bValue		:= p_bOutShutterRetCtrl2;

	END_IF

END_ACTION
```

#### Act_OptP0921OutletShutterFBStat2.st
```iecst
ACTION Act_OptP0921OutletShutterFBStat2:

	tyP0921InletNOutletShutter.tyOutletShutterFB.tyStringStat.sValue	:= p_sOutShutterStatTxt2;

END_ACTION
```

#### Act_OptP0921OutletShutterDC2.st
```iecst
ACTION Act_OptP0921OutletShutterDC2:

	// Direct Control
	IF tyP0921InletNOutletShutter.tyOutletShutterCom2.tyBtnSwitch.bValue = TRUE THEN
		IF p_bOutShutterTwoCtrlOut = FALSE THEN
			IF tyP0921InletNOutletShutter.tyOutletShutterDC2.tyBtnOpen.bRtCompl = TRUE THEN
				tyP0921InletNOutletShutter.tyOutletShutterDC2.tyBtnOpen.bValue	:= TRUE;
				tyP0921InletNOutletShutter.tyOutletShutterDC2.tyBtnClose.bValue	:= FALSE;

				eOutShutterAct2	:= PneuActSetRet;

				IF p_eOutShutterStat2 = PneuActSetRet AND p_eOutShutterStatus2 = Done THEN
					eOutShutterAct2	:= PneuActIdle;

					tyP0921InletNOutletShutter.tyOutletShutterDC2.tyBtnOpen.bRtCompl	:= FALSE;
				END_IF

			ELSIF tyP0921InletNOutletShutter.tyOutletShutterDC2.tyBtnClose.bRtCompl = TRUE THEN
				tyP0921InletNOutletShutter.tyOutletShutterDC2.tyBtnClose.bValue	:= TRUE;
				tyP0921InletNOutletShutter.tyOutletShutterDC2.tyBtnOpen.bValue	:= FALSE;

				eOutShutterAct2	:= PneuActSetExt;

				IF p_eOutShutterStat2 = PneuActSetExt AND p_eOutShutterStatus2 = Done THEN
					eOutShutterAct2	:= PneuActIdle;

					tyP0921InletNOutletShutter.tyOutletShutterDC2.tyBtnClose.bRtCompl	:= FALSE;
				END_IF
			END_IF

		ELSE
			IF (tyP0921InletNOutletShutter.tyOutletShutterDC2.tyBtnOpen.bRtCompl = TRUE) OR (tyP0921InletNOutletShutter.tyOutletShutterDC2.tyBtnClose.bRtCompl = TRUE) THEN
				IF (tyP0921InletNOutletShutter.tyOutletShutterDC2.tyBtnOpen.bValue = TRUE) AND (tyP0921InletNOutletShutter.tyOutletShutterDC2.tyBtnClose.bValue = TRUE) THEN
					eOutShutterAct2	:= PneuActSetAll;

					IF p_eOutShutterStat2 = PneuActSetAll AND p_eOutShutterStatus2 = Done THEN
						eOutShutterAct2	:= PneuActIdle;

						tyP0921InletNOutletShutter.tyOutletShutterDC2.tyBtnOpen.bRtCompl		:= FALSE;
						tyP0921InletNOutletShutter.tyOutletShutterDC2.tyBtnClose.bRtCompl	:= FALSE;
					END_IF

				ELSIF (tyP0921InletNOutletShutter.tyOutletShutterDC2.tyBtnOpen.bValue = TRUE) AND (tyP0921InletNOutletShutter.tyOutletShutterDC2.tyBtnClose.bValue = FALSE) THEN
					eOutShutterAct2	:= PneuActSetRet;

					IF p_eOutShutterStat2 = PneuActSetRet AND p_eOutShutterStatus2 = Done THEN
						eOutShutterAct2	:= PneuActIdle;

						tyP0921InletNOutletShutter.tyOutletShutterDC2.tyBtnOpen.bRtCompl		:= FALSE;
						tyP0921InletNOutletShutter.tyOutletShutterDC2.tyBtnClose.bRtCompl	:= FALSE;
					END_IF

				ELSIF (tyP0921InletNOutletShutter.tyOutletShutterDC2.tyBtnOpen.bValue = FALSE) AND (tyP0921InletNOutletShutter.tyOutletShutterDC2.tyBtnClose.bValue = TRUE) THEN
					eOutShutterAct2	:= PneuActSetExt;

					IF p_eOutShutterStat2 = PneuActSetExt AND p_eOutShutterStatus2 = Done THEN
						eOutShutterAct2	:= PneuActIdle;

						tyP0921InletNOutletShutter.tyOutletShutterDC2.tyBtnOpen.bRtCompl		:= FALSE;
						tyP0921InletNOutletShutter.tyOutletShutterDC2.tyBtnClose.bRtCompl	:= FALSE;
					END_IF

				ELSE
					eOutShutterAct2	:= PneuActRstAll;

					IF p_eOutShutterStat2 = PneuActRstAll AND p_eOutShutterStatus2 = Done THEN
						eOutShutterAct2	:= PneuActIdle;

						tyP0921InletNOutletShutter.tyOutletShutterDC2.tyBtnOpen.bRtCompl		:= FALSE;
						tyP0921InletNOutletShutter.tyOutletShutterDC2.tyBtnClose.bRtCompl	:= FALSE;
					END_IF

				END_IF
			END_IF
		END_IF

		tyP0921InletNOutletShutter.tyOutletShutterFB2.tyBtnOpen.bRtCompl	:= FALSE;
		tyP0921InletNOutletShutter.tyOutletShutterFB2.tyBtnOpen.bValue	:= FALSE;
		tyP0921InletNOutletShutter.tyOutletShutterFB2.tyBtnClose.bRtCompl:= FALSE;
		tyP0921InletNOutletShutter.tyOutletShutterFB2.tyBtnClose.bValue	:= FALSE;

	END_IF

END_ACTION
```

#### Act_EntP0923Disp.st
```iecst
ACTION Act_EntP0923Disp:

	//Access Address
	IF bDispSafetyBar1 = TRUE THEN

		p_tyC0003DualMask ACCESS ADR(tyP0923SafetyBar.tyDualMaskHide);

		IF p_tyNtParamCurr.eProjMag = LDMagDual THEN
			p_tyC0004Navi ACCESS ADR(tyP0923SafetyBar.tyNaviBack);
		ELSE
			p_tyC0004Navi ACCESS ADR(tyP0923SafetyBar.tyNaviLyr1);
		END_IF

		p_tyC0005Main ACCESS ADR(tyCommon.tyMain);

		p_tyC0007Notif ACCESS ADR(tyCommon.tyNotif);

		p_tyC0008MsgBox ACCESS ADR(tyP0923SafetyBar.tyMsgBoxHide);

		p_tyC0009Info ACCESS ADR(tyCommon.tyInfo);

		p_tyP0923LftSafetyBarCom ACCESS ADR(tyP0923SafetyBar.tyMag1SafetyBarCom);
		p_tyP0923LftSafetyBarDC ACCESS ADR(tyP0923SafetyBar.tyMag1SafetyBarDC);
		p_tyP0923LftSafetyBarFB ACCESS ADR(tyP0923SafetyBar.tyMag1SafetyBarFB);

		p_tyP0923RgtSafetyBarCom ACCESS ADR(tyP0923SafetyBar.tyMag2SafetyBarCom);
		p_tyP0923RgtSafetyBarDC ACCESS ADR(tyP0923SafetyBar.tyMag2SafetyBarDC);
		p_tyP0923RgtSafetyBarFB ACCESS ADR(tyP0923SafetyBar.tyMag2SafetyBarFB);

	ELSIF bDispSafetyBar2 = TRUE THEN

		p_tyC0003DualMask ACCESS ADR(tyP0923SafetyBar.tyDualMaskHide);

		p_tyC0004Navi ACCESS ADR(tyP0923SafetyBar.tyNaviLyr2);

		p_tyC0005Main ACCESS ADR(tyCommon.tyMain);

		p_tyC0007Notif ACCESS ADR(tyCommon.tyNotif);

		p_tyC0008MsgBox ACCESS ADR(tyP0923SafetyBar.tyMsgBoxHide);

		p_tyC0009Info ACCESS ADR(tyCommon.tyInfo);

		p_tyP0923LftSafetyBarCom ACCESS ADR(tyP0923SafetyBar.tyMag3SafetyBarCom);
		p_tyP0923LftSafetyBarDC ACCESS ADR(tyP0923SafetyBar.tyMag3SafetyBarDC);
		p_tyP0923LftSafetyBarFB ACCESS ADR(tyP0923SafetyBar.tyMag3SafetyBarFB);

		p_tyP0923RgtSafetyBarCom ACCESS ADR(tyP0923SafetyBar.tyRgtSafetyBarComHide);
		p_tyP0923RgtSafetyBarDC ACCESS ADR(tyP0923SafetyBar.tyRgtSafetyBarDCHide);
		p_tyP0923RgtSafetyBarFB ACCESS ADR(tyP0923SafetyBar.tyRgtSafetyBarFBHide);

	END_IF

	//Disp
	//Update Status
	tyP0923SafetyBar.tyMag1SafetyBarDC.tyBtnExt.bValue	:= p_bMag1SafetyBarExtCtrl;
	tyP0923SafetyBar.tyMag1SafetyBarDC.tyBtnRet.bValue	:= p_bMag1SafetyBarRetCtrl;
	tyP0923SafetyBar.tyMag2SafetyBarDC.tyBtnExt.bValue	:= p_bMag2SafetyBarExtCtrl;
	tyP0923SafetyBar.tyMag2SafetyBarDC.tyBtnRet.bValue	:= p_bMag2SafetyBarRetCtrl;
	tyP0923SafetyBar.tyMag3SafetyBarDC.tyBtnExt.bValue	:= p_bMag3SafetyBarExtCtrl;
	tyP0923SafetyBar.tyMag3SafetyBarDC.tyBtnRet.bValue	:= p_bMag3SafetyBarRetCtrl;

END_ACTION
```

#### Act_OptP0923DualMask.st
```iecst
ACTION Act_OptP0923DualMask:

	IF eCurrPage = UIP0923SafetyBar THEN

		IF p_tyDI.bEStopSig = FALSE THEN
			p_tyC0003DualMask ACCESS ADR(tyP0923SafetyBar.tyDualMaskEStop);

			tyP0923SafetyBar.tyDualMaskEStop.tyBtnLeftMask.uiMaskRtStat.0	:= FALSE;
			tyP0923SafetyBar.tyDualMaskEStop.tyBtnRgtMask.uiMaskRtStat.0	:= bDispSafetyBar2;

		ELSIF p_tyDI.bCoverSWSig = FALSE THEN
			p_tyC0003DualMask ACCESS ADR(tyP0923SafetyBar.tyDualMaskCWSig);

			tyP0923SafetyBar.tyDualMaskCWSig.tyBtnLeftMask.uiMaskRtStat.0	:= FALSE;
			tyP0923SafetyBar.tyDualMaskCWSig.tyBtnRgtMask.uiMaskRtStat.0	:= bDispSafetyBar2;

		ELSIF p_tyDI.bSafetyRlySig = FALSE THEN
			p_tyC0003DualMask ACCESS ADR(tyP0923SafetyBar.tyDualMaskSafetyRly);

			tyP0923SafetyBar.tyDualMaskSafetyRly.tyBtnLeftMask.uiMaskRtStat.0	:= FALSE;
			tyP0923SafetyBar.tyDualMaskSafetyRly.tyBtnRgtMask.uiMaskRtStat.0	:= bDispSafetyBar2;

//		ELSIF p_tyDI.bPullerRetRS = FALSE AND p_tyDI.bInShutterCloseRS = FALSE THEN
//			p_tyC0003DualMask ACCESS ADR(tyP0923SafetyBar.tyDualMaskPshrInterrupt);
//
//			tyP0923SafetyBar.tyDualMaskPshrInterrupt.tyBtnLeftMask.uiMaskRtStat.0	:= FALSE;
//			tyP0923SafetyBar.tyDualMaskPshrInterrupt.tyBtnRgtMask.uiMaskRtStat.0	:= bDispSafetyBar2;

		ELSE
			p_tyC0003DualMask ACCESS ADR(tyP0923SafetyBar.tyDualMaskHide);

		END_IF

	END_IF

END_ACTION
```

#### Act_OptP0923Mag1SafetyBarSen.st
```iecst
ACTION Act_OptP0923Mag1SafetyBarSen:

	tyP0923SafetyBar.tyMag1SafetyBarCom.tyBtnExtRS.bValue	:= p_tyDI.bMag1SafetyBarExtRS;
	tyP0923SafetyBar.tyMag1SafetyBarCom.tyBtnRetRS.bValue	:= p_tyDI.bMag1SafetyBarRetRS;

	//Machine Bitmap
	IF p_tyDI.bMag1SafetyBarRetRS = TRUE THEN
		tyP0923SafetyBar.tyMag1SafetyBarCom.tyBitmapMc.uiValueIdx	:= 1;
	ELSE
		tyP0923SafetyBar.tyMag1SafetyBarCom.tyBitmapMc.uiValueIdx	:= 0;
	END_IF

	IF p_tyNtParamCurr.eProjMag = LDMagTriple AND p_tyNtParamCurr.bProjMotorizedPullerPrep = FALSE THEN
		tyP0923SafetyBar.tyMag1SafetyBarCom.tyBitmapMc.uiValueIdx	:= tyP0923SafetyBar.tyMag1SafetyBarCom.tyBitmapMc.uiValueIdx + 100;
	END_IF

	IF p_tyNtParamCurr.eProjMag = LDMagTriple AND p_tyNtParamCurr.bProjMotorizedPullerPrep = TRUE THEN
		IF 	tyP0923SafetyBar.tyMag1SafetyBarCom.tyBitmapMc.uiValueIdx < 300 THEN
			tyP0923SafetyBar.tyMag1SafetyBarCom.tyBitmapMc.uiValueIdx	:= tyP0923SafetyBar.tyMag1SafetyBarCom.tyBitmapMc.uiValueIdx + 300;
		END_IF
	END_IF
END_ACTION
```

#### Act_OptP0923Mag2SafetyBarSen.st
```iecst
ACTION Act_OptP0923Mag2SafetyBarSen:

	tyP0923SafetyBar.tyMag2SafetyBarCom.tyBtnExtRS.bValue	:= p_tyDI.bMag2SafetyBarExtRS;
	tyP0923SafetyBar.tyMag2SafetyBarCom.tyBtnRetRS.bValue	:= p_tyDI.bMag2SafetyBarRetRS;

	//Machine Bitmap
	IF p_tyDI.bMag2SafetyBarRetRS = TRUE THEN
		tyP0923SafetyBar.tyMag2SafetyBarCom.tyBitmapMc.usiValueIdx	:= 3;
	ELSE
		tyP0923SafetyBar.tyMag2SafetyBarCom.tyBitmapMc.usiValueIdx	:= 2;
	END_IF

	IF p_tyNtParamCurr.eProjMag = LDMagTriple AND p_tyNtParamCurr.bProjMotorizedPullerPrep = FALSE THEN
		tyP0923SafetyBar.tyMag2SafetyBarCom.tyBitmapMc.uiValueIdx	:= tyP0923SafetyBar.tyMag2SafetyBarCom.tyBitmapMc.uiValueIdx + 100;
	END_IF

	IF p_tyNtParamCurr.eProjMag = LDMagTriple AND p_tyNtParamCurr.bProjMotorizedPullerPrep = TRUE THEN
			IF 	tyP0923SafetyBar.tyMag2SafetyBarCom.tyBitmapMc.uiValueIdx < 300 THEN
				tyP0923SafetyBar.tyMag2SafetyBarCom.tyBitmapMc.uiValueIdx	:= tyP0923SafetyBar.tyMag2SafetyBarCom.tyBitmapMc.uiValueIdx + 300;
			END_IF
	END_IF

END_ACTION
```

#### Act_OptP0923Mag3SafetyBarSen.st
```iecst
ACTION Act_OptP0923Mag3SafetyBarSen:

	tyP0923SafetyBar.tyMag3SafetyBarCom.tyBtnExtRS.bValue	:= p_tyDI.bMag3SafetyBarExtRS;
	tyP0923SafetyBar.tyMag3SafetyBarCom.tyBtnRetRS.bValue	:= p_tyDI.bMag3SafetyBarRetRS;

	//Machine Bitmap
	IF p_tyDI.bMag3SafetyBarRetRS = TRUE THEN
		tyP0923SafetyBar.tyMag3SafetyBarCom.tyBitmapMc.usiValueIdx	:= 5;
	ELSE
		tyP0923SafetyBar.tyMag3SafetyBarCom.tyBitmapMc.usiValueIdx	:= 4;
	END_IF

	IF p_tyNtParamCurr.eProjMag = LDMagTriple AND p_tyNtParamCurr.bProjMotorizedPullerPrep = FALSE THEN
		tyP0923SafetyBar.tyMag3SafetyBarCom.tyBitmapMc.uiValueIdx	:= tyP0923SafetyBar.tyMag3SafetyBarCom.tyBitmapMc.uiValueIdx + 100;
	END_IF

	IF p_tyNtParamCurr.eProjMag = LDMagTriple AND p_tyNtParamCurr.bProjMotorizedPullerPrep = TRUE THEN
			IF 	tyP0923SafetyBar.tyMag3SafetyBarCom.tyBitmapMc.uiValueIdx < 300 THEN
				tyP0923SafetyBar.tyMag3SafetyBarCom.tyBitmapMc.uiValueIdx	:= tyP0923SafetyBar.tyMag3SafetyBarCom.tyBitmapMc.uiValueIdx + 300;
			END_IF
	END_IF

END_ACTION
```

#### Act_OptP0923Navi.st
```iecst
ACTION Act_OptP0923Navi:

	IF tyP0923SafetyBar.tyNaviBack.tyBtnBack.bRtCompl = TRUE OR tyP0923SafetyBar.tyNaviLyr1.tyBtnBack.bRtCompl = TRUE OR tyP0923SafetyBar.tyNaviLyr2.tyBtnBack.bRtCompl = TRUE THEN
		tyP0923SafetyBar.tyNaviBack.tyBtnBack.bRtCompl 	:= FALSE;
		tyP0923SafetyBar.tyNaviBack.tyBtnBack.bValue	:= FALSE;
		tyP0923SafetyBar.tyNaviLyr1.tyBtnBack.bRtCompl 	:= FALSE;
		tyP0923SafetyBar.tyNaviLyr1.tyBtnBack.bValue	:= FALSE;
		tyP0923SafetyBar.tyNaviLyr2.tyBtnBack.bRtCompl 	:= FALSE;
		tyP0923SafetyBar.tyNaviLyr2.tyBtnBack.bValue	:= FALSE;

		eChgPage	:= UIP0920MtrNPneuCtrl;

	ELSIF tyP0923SafetyBar.tyNaviLyr1.tyBtnLeft.bRtCompl = TRUE OR tyP0923SafetyBar.tyNaviLyr1.tyBtnRgt.bRtCompl = TRUE THEN
		tyP0923SafetyBar.tyNaviLyr1.tyBtnLeft.bRtCompl	:= FALSE;
		tyP0923SafetyBar.tyNaviLyr1.tyBtnRgt.bRtCompl	:= FALSE;

		bDispSafetyBar1	:= FALSE;
		bDispSafetyBar2	:= TRUE;

		p_tyC0004Navi ACCESS ADR(tyP0923SafetyBar.tyNaviLyr2);

		p_tyP0923LftSafetyBarCom ACCESS ADR(tyP0923SafetyBar.tyMag3SafetyBarCom);
		p_tyP0923LftSafetyBarDC ACCESS ADR(tyP0923SafetyBar.tyMag3SafetyBarDC);
		p_tyP0923LftSafetyBarFB ACCESS ADR(tyP0923SafetyBar.tyMag3SafetyBarFB);

		p_tyP0923RgtSafetyBarCom ACCESS ADR(tyP0923SafetyBar.tyRgtSafetyBarComHide);
		p_tyP0923RgtSafetyBarDC ACCESS ADR(tyP0923SafetyBar.tyRgtSafetyBarDCHide);
		p_tyP0923RgtSafetyBarFB ACCESS ADR(tyP0923SafetyBar.tyRgtSafetyBarFBHide);

	ELSIF tyP0923SafetyBar.tyNaviLyr2.tyBtnLeft.bRtCompl = TRUE OR tyP0923SafetyBar.tyNaviLyr2.tyBtnRgt.bRtCompl = TRUE THEN
		tyP0923SafetyBar.tyNaviLyr2.tyBtnLeft.bRtCompl	:= FALSE;
		tyP0923SafetyBar.tyNaviLyr2.tyBtnRgt.bRtCompl	:= FALSE;

		bDispSafetyBar1	:= TRUE;
		bDispSafetyBar2	:= FALSE;

		p_tyC0004Navi ACCESS ADR(tyP0923SafetyBar.tyNaviLyr1);

		p_tyP0923LftSafetyBarCom ACCESS ADR(tyP0923SafetyBar.tyMag1SafetyBarCom);
		p_tyP0923LftSafetyBarDC ACCESS ADR(tyP0923SafetyBar.tyMag1SafetyBarDC);
		p_tyP0923LftSafetyBarFB ACCESS ADR(tyP0923SafetyBar.tyMag1SafetyBarFB);

		p_tyP0923RgtSafetyBarCom ACCESS ADR(tyP0923SafetyBar.tyMag2SafetyBarCom);
		p_tyP0923RgtSafetyBarDC ACCESS ADR(tyP0923SafetyBar.tyMag2SafetyBarDC);
		p_tyP0923RgtSafetyBarFB ACCESS ADR(tyP0923SafetyBar.tyMag2SafetyBarFB);

	END_IF

END_ACTION
```

#### Act_OptP0923RstMnl.st
```iecst
ACTION Act_OptP0923RstMnl:

	IF EDGEPOS((bManualMod = FALSE) OR (p_eMag1SafetyBarStatus = Error)) THEN

		eMag1SafetyBarAct	:= PneuActIdle;

		tyP0923SafetyBar.tyMag1SafetyBarDC.tyBtnRet.bRtCompl	:= FALSE;
		tyP0923SafetyBar.tyMag1SafetyBarDC.tyBtnRet.bValue		:= FALSE;
		tyP0923SafetyBar.tyMag1SafetyBarDC.tyBtnExt.bRtCompl	:= FALSE;
		tyP0923SafetyBar.tyMag1SafetyBarDC.tyBtnExt.bValue		:= FALSE;

		tyP0923SafetyBar.tyMag1SafetyBarFB.tyBtnRet.bRtCompl	:= FALSE;
		tyP0923SafetyBar.tyMag1SafetyBarFB.tyBtnRet.bValue		:= FALSE;
		tyP0923SafetyBar.tyMag1SafetyBarFB.tyBtnExt.bRtCompl	:= FALSE;
		tyP0923SafetyBar.tyMag1SafetyBarFB.tyBtnExt.bValue		:= FALSE;

	END_IF

	IF EDGEPOS((bManualMod = FALSE) OR (p_eMag2SafetyBarStatus = Error)) THEN

		eMag2SafetyBarAct	:= PneuActIdle;

		tyP0923SafetyBar.tyMag2SafetyBarDC.tyBtnRet.bRtCompl	:= FALSE;
		tyP0923SafetyBar.tyMag2SafetyBarDC.tyBtnRet.bValue		:= FALSE;
		tyP0923SafetyBar.tyMag2SafetyBarDC.tyBtnExt.bRtCompl	:= FALSE;
		tyP0923SafetyBar.tyMag2SafetyBarDC.tyBtnExt.bValue		:= FALSE;

		tyP0923SafetyBar.tyMag2SafetyBarFB.tyBtnRet.bRtCompl	:= FALSE;
		tyP0923SafetyBar.tyMag2SafetyBarFB.tyBtnRet.bValue		:= FALSE;
		tyP0923SafetyBar.tyMag2SafetyBarFB.tyBtnExt.bRtCompl	:= FALSE;
		tyP0923SafetyBar.tyMag2SafetyBarFB.tyBtnExt.bValue		:= FALSE;

	END_IF

	IF EDGEPOS((bManualMod = FALSE) OR (p_eMag3SafetyBarStatus = Error)) THEN

		eMag3SafetyBarAct	:= PneuActIdle;

		tyP0923SafetyBar.tyMag3SafetyBarDC.tyBtnRet.bRtCompl	:= FALSE;
		tyP0923SafetyBar.tyMag3SafetyBarDC.tyBtnRet.bValue		:= FALSE;
		tyP0923SafetyBar.tyMag3SafetyBarDC.tyBtnExt.bRtCompl	:= FALSE;
		tyP0923SafetyBar.tyMag3SafetyBarDC.tyBtnExt.bValue		:= FALSE;

		tyP0923SafetyBar.tyMag3SafetyBarFB.tyBtnRet.bRtCompl	:= FALSE;
		tyP0923SafetyBar.tyMag3SafetyBarFB.tyBtnRet.bValue		:= FALSE;
		tyP0923SafetyBar.tyMag3SafetyBarFB.tyBtnExt.bRtCompl	:= FALSE;
		tyP0923SafetyBar.tyMag3SafetyBarFB.tyBtnExt.bValue		:= FALSE;

	END_IF

END_ACTION
```

#### Act_EntP0924Disp.st
```iecst
ACTION Act_EntP0924Disp:

	//Access Address
	p_tyC0002FullMask ACCESS ADR(tyP0924TrolleyLck.tyFullMaskHide);

	p_tyC0004Navi ACCESS ADR(tyP0924TrolleyLck.tyNaviBack);

	p_tyC0005Main ACCESS ADR(tyCommon.tyMain);

	p_tyC0007Notif ACCESS ADR(tyCommon.tyNotif);

	p_tyC0008MsgBox ACCESS ADR(tyP0924TrolleyLck.tyMsgBoxHide);

	p_tyC0009Info ACCESS ADR(tyCommon.tyInfo);

	p_tyP0924TrolleyLckCom ACCESS ADR(tyP0924TrolleyLck.tyCom);
	p_tyP0924TrolleyLckDC ACCESS ADR(tyP0924TrolleyLck.tyDC);
	p_tyP0924TrolleyLckFB ACCESS ADR(tyP0924TrolleyLck.tyFB);

	IF tyP0924TrolleyLck.tyCom.tyBtnSwitch.bValue THEN
		fUIInRtStatHide(ADR(tyP0924TrolleyLck.tyFB.tyLyr.uiRtStat));
		fUIInRtStatOff(ADR(tyP0924TrolleyLck.tyDC.tyLyr.uiRtStat));
	ELSE
		fUIInRtStatOff(ADR(tyP0924TrolleyLck.tyFB.tyLyr.uiRtStat));
		fUIInRtStatHide(ADR(tyP0924TrolleyLck.tyDC.tyLyr.uiRtStat));
	END_IF

END_ACTION
```

#### Act_OptP0924FullMask.st
```iecst
ACTION Act_OptP0924FullMask:

	IF eCurrPage = UIP0924TrolleyLck THEN

		IF p_tyDI.bEStopSig = FALSE THEN
			p_tyC0002FullMask ACCESS ADR(tyP0924TrolleyLck.tyFullMaskEStop);

		ELSIF p_tyDI.bCoverSWSig = FALSE THEN
			p_tyC0002FullMask ACCESS ADR(tyP0924TrolleyLck.tyFullMaskCWSig);

		ELSIF p_tyDI.bSafetyRlySig = FALSE THEN
			p_tyC0002FullMask ACCESS ADR(tyP0924TrolleyLck.tyFullMaskSafetyRly);

		ELSE
			p_tyC0002FullMask ACCESS ADR(tyP0924TrolleyLck.tyFullMaskHide);

		END_IF

	END_IF

END_ACTION
```

#### Act_OptP0924Navi.st
```iecst
ACTION Act_OptP0924Navi:

	IF tyP0924TrolleyLck.tyNaviBack.tyBtnBack.bRtCompl = TRUE THEN
		tyP0924TrolleyLck.tyNaviBack.tyBtnBack.bRtCompl	:= FALSE;
		tyP0924TrolleyLck.tyNaviBack.tyBtnBack.bValue	:= FALSE;
		eChgPage	:= UIP0920MtrNPneuCtrl;
	END_IF

END_ACTION
```

#### Act_OptP0924TrolleyLckChgLyr.st
```iecst
ACTION Act_OptP0924TrolleyLckChgLyr:

	IF tyP0924TrolleyLck.tyCom.tyBtnSwitch.bRtCompl THEN
		tyP0924TrolleyLck.tyCom.tyBtnSwitch.bRtCompl	:= FALSE;

		IF tyP0924TrolleyLck.tyCom.tyBtnSwitch.bValue = TRUE THEN
			fUIInRtStatOff(ADR(tyP0924TrolleyLck.tyDC.tyLyr.uiRtStat));
			fUIInRtStatHide(ADR(tyP0924TrolleyLck.tyFB.tyLyr.uiRtStat));
		ELSE
			fUIInRtStatHide(ADR(tyP0924TrolleyLck.tyDC.tyLyr.uiRtStat));
			fUIInRtStatOff(ADR(tyP0924TrolleyLck.tyFB.tyLyr.uiRtStat));
		END_IF

	END_IF

END_ACTION
```

#### Act_OptP0924TrolleyLckSen.st
```iecst
ACTION Act_OptP0924TrolleyLckSen:

	tyP0924TrolleyLck.tyCom.tyBtnExtRS.bValue			:= p_tyDI.bTrolleyExtRS1;
	tyP0924TrolleyLck.tyCom.tyBtnExtRS2.bValue			:= p_tyDI.bTrolleyExtRS2;
	tyP0924TrolleyLck.tyCom.tyBtnPresentSen1.bValue			:= p_tyDI.bTrolleyPreSen1;
	tyP0924TrolleyLck.tyCom.tyBtnPresentSen2.bValue			:= p_tyDI.bTrolleyPreSen2;

	//Bitmap default: 456 mag1
	IF   (p_tyNtParamCurr.eProjMag = LDMagDual AND p_tyNtParamCurr.bMagAutoVerifyPrep = FALSE)
		OR (p_tyNtParamCurr.eProjMag = LDMagTriple AND p_tyNtParamCurr.bMagAutoVerifyPrep = FALSE)
		OR (p_tyNtParamCurr.eProjMag = LDMagDual AND p_tyNtParamCurr.bMagAutoVerifyPrep = TRUE)
		THEN
		IF eTrolleyLckAct1 = PneuActExt OR eTrolleyLckAct1 = PneuActRet OR
			eTrolleyLckAct1 = PneuActSetExt OR eTrolleyLckAct1 = PneuActSetRet THEN
			tyP0924TrolleyLck.tyCom.tyBitmapMc.usiValueIdx := 0;
		ELSIF eTrolleyLckAct2 = PneuActExt OR eTrolleyLckAct2 = PneuActRet OR
			eTrolleyLckAct2 = PneuActSetExt	OR eTrolleyLckAct2 = PneuActSetRet THEN
			tyP0924TrolleyLck.tyCom.tyBitmapMc.usiValueIdx := 1;
		END_IF
	END_IF

END_ACTION
```

#### Act_OptP0924TrolleyLckFB.st
```iecst
ACTION Act_OptP0924TrolleyLckFB:

	IF tyP0924TrolleyLck.tyCom.tyBtnSwitch.bValue = FALSE THEN

		IF tyP0924TrolleyLck.tyFB.tyBtnRet.bRtCompl = TRUE THEN
			tyP0924TrolleyLck.tyFB.tyBtnRet.bRtCompl	:= FALSE;

			tyP0924TrolleyLck.tyFB.tyBtnRet.bValue		:= TRUE;
			tyP0924TrolleyLck.tyFB.tyBtnExt.bValue		:= FALSE;

		ELSIF tyP0924TrolleyLck.tyFB.tyBtnExt.bRtCompl = TRUE THEN
			tyP0924TrolleyLck.tyFB.tyBtnExt.bRtCompl	:= FALSE;

			tyP0924TrolleyLck.tyFB.tyBtnExt.bValue		:= TRUE;
			tyP0924TrolleyLck.tyFB.tyBtnRet.bValue		:= FALSE;

		ELSIF tyP0924TrolleyLck.tyFB.tyBtnRet2.bRtCompl = TRUE THEN
			tyP0924TrolleyLck.tyFB.tyBtnRet2.bRtCompl	:= FALSE;

			tyP0924TrolleyLck.tyFB.tyBtnRet2.bValue		:= TRUE;
			tyP0924TrolleyLck.tyFB.tyBtnExt2.bValue		:= FALSE;

		ELSIF tyP0924TrolleyLck.tyFB.tyBtnExt2.bRtCompl = TRUE THEN
			tyP0924TrolleyLck.tyFB.tyBtnExt2.bRtCompl	:= FALSE;

			tyP0924TrolleyLck.tyFB.tyBtnExt2.bValue		:= TRUE;
			tyP0924TrolleyLck.tyFB.tyBtnRet2.bValue		:= FALSE;
		END_IF

		IF tyP0924TrolleyLck.tyFB.tyBtnRet.bValue = TRUE THEN
			//Trolley lock mag 1
			eTrolleyLckAct1	:= PneuActRet;

			IF p_eTrolleyLckStat = PneuActRet AND p_eTrolleyLckStatus = Done THEN
				eTrolleyLckAct1	:= PneuActIdle;
				tyP0924TrolleyLck.tyFB.tyBtnRet.bValue	:= FALSE;
			ELSIF p_eTrolleyLckStatus = Error THEN
				tyP0924TrolleyLck.tyFB.tyBtnRet.bValue	:= FALSE;
			END_IF

		ELSIF tyP0924TrolleyLck.tyFB.tyBtnExt.bValue = TRUE THEN
			eTrolleyLckAct1	:= PneuActExt;

			IF p_eTrolleyLckStat = PneuActExt AND p_eTrolleyLckStatus = Done THEN
				eTrolleyLckAct1	:= PneuActIdle;
				tyP0924TrolleyLck.tyFB.tyBtnExt.bValue := FALSE;
			ELSIF p_eTrolleyLckStatus = Error THEN
				tyP0924TrolleyLck.tyFB.tyBtnExt.bValue := FALSE;
			END_IF

		ELSIF tyP0924TrolleyLck.tyFB.tyBtnRet2.bValue = TRUE THEN
			//Trolley lock Mag 2
			eTrolleyLckAct2	:= PneuActRet;

			IF p_eTrolleyLckStat2 = PneuActRet AND p_eTrolleyLckStatus2 = Done THEN
				eTrolleyLckAct2	:= PneuActIdle;
				tyP0924TrolleyLck.tyFB.tyBtnRet2.bValue	:= FALSE;
			ELSIF p_eTrolleyLckStatus2 = Error THEN
				tyP0924TrolleyLck.tyFB.tyBtnRet2.bValue	:= FALSE;
			END_IF

		ELSIF tyP0924TrolleyLck.tyFB.tyBtnExt2.bValue = TRUE THEN
			eTrolleyLckAct2	:= PneuActExt;

			IF p_eTrolleyLckStat2 = PneuActExt AND p_eTrolleyLckStatus2 = Done THEN
				eTrolleyLckAct2	:= PneuActIdle;
				tyP0924TrolleyLck.tyFB.tyBtnExt2.bValue := FALSE;
			ELSIF p_eTrolleyLckStatus2 = Error THEN
				tyP0924TrolleyLck.tyFB.tyBtnExt2.bValue := FALSE;
			END_IF
		END_IF

		//Update Direct Control Status
		tyP0924TrolleyLck.tyDC.tyBtnRet.bRtCompl	:= FALSE;
		tyP0924TrolleyLck.tyDC.tyBtnExt.bRtCompl	:= FALSE;
		tyP0924TrolleyLck.tyDC.tyBtnRet.bValue		:= p_bTrolleyLckRetCtrl;
		tyP0924TrolleyLck.tyDC.tyBtnExt.bValue		:= p_bTrolleyLckExtCtrl;

		tyP0924TrolleyLck.tyDC.tyBtnRet2.bRtCompl	:= FALSE;
		tyP0924TrolleyLck.tyDC.tyBtnExt2.bRtCompl	:= FALSE;
		tyP0924TrolleyLck.tyDC.tyBtnRet2.bValue		:= p_bTrolleyLckRetCtrl2;
		tyP0924TrolleyLck.tyDC.tyBtnExt2.bValue		:= p_bTrolleyLckExtCtrl2;

	END_IF

END_ACTION
```

#### Act_OptP0924TrolleyLckFBStat.st
```iecst
ACTION Act_OptP0924TrolleyLckFBStat:
	IF tyP0924TrolleyLck.tyFB.tyBtnRet.bValue OR tyP0924TrolleyLck.tyFB.tyBtnExt.bValue OR
		tyP0924TrolleyLck.tyDC.tyBtnRet.bValue OR tyP0924TrolleyLck.tyDC.tyBtnExt.bValue THEN

		tyP0924TrolleyLck.tyFB.tyStringStat.sValue	:= p_sTrolleyLckStatTxt;

	ELSIF tyP0924TrolleyLck.tyFB.tyBtnRet2.bValue OR tyP0924TrolleyLck.tyFB.tyBtnExt2.bValue OR
		tyP0924TrolleyLck.tyDC.tyBtnRet2.bValue OR tyP0924TrolleyLck.tyDC.tyBtnExt2.bValue THEN

		tyP0924TrolleyLck.tyFB.tyStringStat.sValue	:= p_sTrolleyLckStatTxt2;
	ELSE
		tyP0924TrolleyLck.tyFB.tyStringStat.sValue	:= p_sTrolleyLckStatTxt;

	END_IF

END_ACTION
```

#### Act_OptP0924TrolleyLckDC.st
```iecst
ACTION Act_OptP0924TrolleyLckDC:

	IF tyP0924TrolleyLck.tyCom.tyBtnSwitch.bValue = TRUE THEN

		IF p_bTrolleyLckTwoCtrlOut = FALSE THEN

			IF tyP0924TrolleyLck.tyDC.tyBtnRet.bRtCompl = TRUE THEN
				tyP0924TrolleyLck.tyDC.tyBtnRet.bValue	:= TRUE;
				tyP0924TrolleyLck.tyDC.tyBtnExt.bValue	:= FALSE;

				eTrolleyLckAct1	:= PneuActSetRet; //4

				IF p_eTrolleyLckStat = PneuActSetRet AND p_eTrolleyLckStatus = Done THEN
					eTrolleyLckAct1	:= PneuActIdle;

					tyP0924TrolleyLck.tyDC.tyBtnRet.bRtCompl	:= FALSE;
				END_IF

			ELSIF tyP0924TrolleyLck.tyDC.tyBtnExt.bRtCompl = TRUE THEN
				tyP0924TrolleyLck.tyDC.tyBtnExt.bValue	:= TRUE;
				tyP0924TrolleyLck.tyDC.tyBtnRet.bValue	:= FALSE;

				eTrolleyLckAct1	:= PneuActSetExt; //3

				IF p_eTrolleyLckStat = PneuActSetExt AND p_eTrolleyLckStatus = Done THEN
					eTrolleyLckAct1	:= PneuActIdle;

					tyP0924TrolleyLck.tyDC.tyBtnExt.bRtCompl	:= FALSE;
				END_IF

			ELSIF tyP0924TrolleyLck.tyDC.tyBtnRet2.bRtCompl = TRUE THEN
				tyP0924TrolleyLck.tyDC.tyBtnRet2.bValue	:= TRUE;
				tyP0924TrolleyLck.tyDC.tyBtnExt2.bValue	:= FALSE;

				eTrolleyLckAct2	:= PneuActSetRet; //4

				IF p_eTrolleyLckStat2 = PneuActSetRet AND p_eTrolleyLckStatus2 = Done THEN
					eTrolleyLckAct2	:= PneuActIdle;

					tyP0924TrolleyLck.tyDC.tyBtnRet2.bRtCompl	:= FALSE;
				END_IF

			ELSIF tyP0924TrolleyLck.tyDC.tyBtnExt2.bRtCompl = TRUE THEN
				tyP0924TrolleyLck.tyDC.tyBtnExt2.bValue	:= TRUE;
				tyP0924TrolleyLck.tyDC.tyBtnRet2.bValue	:= FALSE;

				eTrolleyLckAct2	:= PneuActSetExt; //3

				IF p_eTrolleyLckStat2 = PneuActSetExt AND p_eTrolleyLckStatus2 = Done THEN
					eTrolleyLckAct2	:= PneuActIdle;

					tyP0924TrolleyLck.tyDC.tyBtnExt2.bRtCompl	:= FALSE;
				END_IF
			END_IF

		ELSE
			//Trolley 1---------------
			IF (tyP0924TrolleyLck.tyDC.tyBtnRet.bRtCompl = TRUE) OR (tyP0924TrolleyLck.tyDC.tyBtnExt.bRtCompl = TRUE) THEN

				IF (tyP0924TrolleyLck.tyDC.tyBtnRet.bValue = TRUE) AND (tyP0924TrolleyLck.tyDC.tyBtnExt.bValue = TRUE) THEN
					eTrolleyLckAct1	:= PneuActSetAll;

					IF p_eTrolleyLckStat = PneuActSetAll AND p_eTrolleyLckStatus = Done THEN
						eTrolleyLckAct1	:= PneuActIdle;

						tyP0924TrolleyLck.tyDC.tyBtnRet.bRtCompl	:= FALSE;
						tyP0924TrolleyLck.tyDC.tyBtnExt.bRtCompl	:= FALSE;
					END_IF

				ELSIF (tyP0924TrolleyLck.tyDC.tyBtnRet.bValue = TRUE) AND (tyP0924TrolleyLck.tyDC.tyBtnExt.bValue = FALSE) THEN
					eTrolleyLckAct1	:= PneuActSetRet;

					IF p_eTrolleyLckStat = PneuActSetRet AND p_eTrolleyLckStatus = Done THEN
						eTrolleyLckAct1	:= PneuActIdle;

						tyP0924TrolleyLck.tyDC.tyBtnRet.bRtCompl	:= FALSE;
						tyP0924TrolleyLck.tyDC.tyBtnExt.bRtCompl	:= FALSE;
					END_IF

				ELSIF (tyP0924TrolleyLck.tyDC.tyBtnRet.bValue = FALSE) AND (tyP0924TrolleyLck.tyDC.tyBtnExt.bValue = TRUE) THEN
					eTrolleyLckAct1	:= PneuActSetExt;

					IF p_eTrolleyLckStat = PneuActSetExt AND p_eTrolleyLckStatus = Done THEN
						eTrolleyLckAct1	:= PneuActIdle;

						tyP0924TrolleyLck.tyDC.tyBtnRet.bRtCompl	:= FALSE;
						tyP0924TrolleyLck.tyDC.tyBtnExt.bRtCompl	:= FALSE;
					END_IF

				ELSE
					eTrolleyLckAct1	:= PneuActRstAll;

					IF p_eTrolleyLckStat = PneuActRstAll AND p_eTrolleyLckStatus = Done THEN
						eTrolleyLckAct1	:= PneuActIdle;

						tyP0924TrolleyLck.tyDC.tyBtnRet.bRtCompl	:= FALSE;
						tyP0924TrolleyLck.tyDC.tyBtnExt.bRtCompl	:= FALSE;
					END_IF

				END_IF

			END_IF
			//Trolley 2---------------
			IF (tyP0924TrolleyLck.tyDC.tyBtnRet2.bRtCompl = TRUE) OR (tyP0924TrolleyLck.tyDC.tyBtnExt2.bRtCompl = TRUE) THEN

				IF (tyP0924TrolleyLck.tyDC.tyBtnRet2.bValue = TRUE) AND (tyP0924TrolleyLck.tyDC.tyBtnExt2.bValue = TRUE) THEN
					eTrolleyLckAct2	:= PneuActSetAll;

					IF p_eTrolleyLckStat2 = PneuActSetAll AND p_eTrolleyLckStatus2 = Done THEN
						eTrolleyLckAct2	:= PneuActIdle;

						tyP0924TrolleyLck.tyDC.tyBtnRet2.bRtCompl	:= FALSE;
						tyP0924TrolleyLck.tyDC.tyBtnExt2.bRtCompl	:= FALSE;
					END_IF

				ELSIF (tyP0924TrolleyLck.tyDC.tyBtnRet2.bValue = TRUE) AND (tyP0924TrolleyLck.tyDC.tyBtnExt2.bValue = FALSE) THEN
					eTrolleyLckAct2	:= PneuActSetRet;

					IF p_eTrolleyLckStat2 = PneuActSetRet AND p_eTrolleyLckStatus2 = Done THEN
						eTrolleyLckAct2	:= PneuActIdle;

						tyP0924TrolleyLck.tyDC.tyBtnRet2.bRtCompl	:= FALSE;
						tyP0924TrolleyLck.tyDC.tyBtnExt2.bRtCompl	:= FALSE;
					END_IF

				ELSIF (tyP0924TrolleyLck.tyDC.tyBtnRet2.bValue = FALSE) AND (tyP0924TrolleyLck.tyDC.tyBtnExt2.bValue = TRUE) THEN
					eTrolleyLckAct2	:= PneuActSetExt;

					IF p_eTrolleyLckStat2 = PneuActSetExt AND p_eTrolleyLckStatus2 = Done THEN
						eTrolleyLckAct2	:= PneuActIdle;

						tyP0924TrolleyLck.tyDC.tyBtnRet2.bRtCompl	:= FALSE;
						tyP0924TrolleyLck.tyDC.tyBtnExt2.bRtCompl	:= FALSE;
					END_IF

				ELSE
					eTrolleyLckAct2	:= PneuActRstAll;

					IF p_eTrolleyLckStat2 = PneuActRstAll AND p_eTrolleyLckStatus2 = Done THEN
						eTrolleyLckAct2	:= PneuActIdle;

						tyP0924TrolleyLck.tyDC.tyBtnRet2.bRtCompl	:= FALSE;
						tyP0924TrolleyLck.tyDC.tyBtnExt2.bRtCompl	:= FALSE;
					END_IF

				END_IF

			END_IF
		END_IF

		tyP0924TrolleyLck.tyFB.tyBtnExt.bRtCompl	:= FALSE;
		tyP0924TrolleyLck.tyFB.tyBtnExt.bValue		:= FALSE;
		tyP0924TrolleyLck.tyFB.tyBtnRet.bRtCompl	:= FALSE;
		tyP0924TrolleyLck.tyFB.tyBtnRet.bValue		:= FALSE;

		tyP0924TrolleyLck.tyFB.tyBtnExt2.bRtCompl	:= FALSE;
		tyP0924TrolleyLck.tyFB.tyBtnExt2.bValue		:= FALSE;
		tyP0924TrolleyLck.tyFB.tyBtnRet2.bRtCompl	:= FALSE;
		tyP0924TrolleyLck.tyFB.tyBtnRet2.bValue		:= FALSE;

	END_IF

END_ACTION
```

#### Act_OptP0924RstMnl.st
```iecst
ACTION Act_OptP0924RstMnl:

	IF EDGEPOS((bManualMod = FALSE) OR (p_eTrolleyLckStatus = Error)) THEN

		eTrolleyLckAct1	:= PneuActIdle;

		tyP0924TrolleyLck.tyDC.tyBtnRet.bRtCompl	:= FALSE;
		tyP0924TrolleyLck.tyDC.tyBtnRet.bValue		:= FALSE;
		tyP0924TrolleyLck.tyDC.tyBtnExt.bRtCompl	:= FALSE;
		tyP0924TrolleyLck.tyDC.tyBtnExt.bValue		:= FALSE;

		tyP0924TrolleyLck.tyFB.tyBtnRet.bRtCompl	:= FALSE;
		tyP0924TrolleyLck.tyFB.tyBtnRet.bValue		:= FALSE;
		tyP0924TrolleyLck.tyFB.tyBtnExt.bRtCompl	:= FALSE;
		tyP0924TrolleyLck.tyFB.tyBtnExt.bValue		:= FALSE;

	END_IF

	IF EDGEPOS((bManualMod = FALSE) OR (p_eTrolleyLckStatus2 = Error)) THEN

		eTrolleyLckAct2	:= PneuActIdle;

		tyP0924TrolleyLck.tyDC.tyBtnRet2.bRtCompl	:= FALSE;
		tyP0924TrolleyLck.tyDC.tyBtnRet2.bValue		:= FALSE;
		tyP0924TrolleyLck.tyDC.tyBtnExt2.bRtCompl	:= FALSE;
		tyP0924TrolleyLck.tyDC.tyBtnExt2.bValue		:= FALSE;

		tyP0924TrolleyLck.tyFB.tyBtnRet2.bRtCompl	:= FALSE;
		tyP0924TrolleyLck.tyFB.tyBtnRet2.bValue		:= FALSE;
		tyP0924TrolleyLck.tyFB.tyBtnExt2.bRtCompl	:= FALSE;
		tyP0924TrolleyLck.tyFB.tyBtnExt2.bValue		:= FALSE;

	END_IF

END_ACTION
```

#### Act_EntP0930Disp.st
```iecst
ACTION Act_EntP0930Disp:

	//Access Address
	p_tyC0002FullMask ACCESS ADR(tyP0930MagConv1.tyFullMaskHide);

//	p_tyC0004Navi ACCESS ADR(tyP0930MagConv1.tyNaviBack);
	CASE p_tyNtParamCurr.eProjMag OF
		LDMagDual:
			p_tyC0004Navi ACCESS ADR(tyP0930MagConv1.tyNavi2Lyr1);
		LDMagTriple:
			p_tyC0004Navi ACCESS ADR(tyP0930MagConv1.tyNavi3Lyr1);
		LDMagQuadruple:
			p_tyC0004Navi ACCESS ADR(tyP0930MagConv1.tyNavi4Lyr1);
	END_CASE

	p_tyC0005Main ACCESS ADR(tyCommon.tyMain);

	p_tyC0007Notif ACCESS ADR(tyCommon.tyNotif);

	p_tyC0008MsgBox ACCESS ADR(tyP0930MagConv1.tyMsgBoxHide);

	p_tyC0009Info ACCESS ADR(tyCommon.tyInfo);

	p_tyP0930Mag1ConvCom ACCESS ADR(tyP0930MagConv1.tyCom);
	p_tyP0930Mag1ConvDC ACCESS ADR(tyP0930MagConv1.tyDC);
	p_tyP0930Mag1ConvFB ACCESS ADR(tyP0930MagConv1.tyFB);

	IF p_tyNtParamCurr.eProjMag = LDMagDual AND p_tyNtParamCurr.bMagAutoVerifyPrep = FALSE THEN
		tyP0930MagConv1.tyCom.tyBitmapMc.usiValueIdx	:= 142;
	ELSIF p_tyNtParamCurr.eProjMag = LDMagDual AND p_tyNtParamCurr.bMagAutoVerifyPrep = TRUE THEN
		tyP0930MagConv1.tyCom.tyBitmapMc.usiValueIdx	:= 200;
	ELSIF p_tyNtParamCurr.eProjMag = LDMagTriple AND p_tyNtParamCurr.bMagAutoVerifyPrep = TRUE THEN
		tyP0930MagConv1.tyCom.tyBitmapMc.usiValueIdx	:= 0;
	ELSIF p_tyNtParamCurr.eProjMag = LDMagQuadruple AND p_tyNtParamCurr.bMagAutoVerifyPrep = TRUE THEN
		tyP0930MagConv1.tyCom.tyBitmapMc.usiValueIdx	:= 66;
	ELSE
		tyP0930MagConv1.tyCom.tyBitmapMc.usiValueIdx	:= 100;
	END_IF

	IF p_tyNtParamCurr.bMagAutoVerifyPrep = FALSE THEN
		tyP0930MagConv1.tyFB.tyBtnFixedClamp.usiTxtIdx	:= 6;
		tyP0930MagConv1.tyFB.tyBtnFixedUnclamp.usiTxtIdx:= 6;
		tyP0930MagConv1.tyFB.tyBtnRemoteClamp.usiTxtIdx	:= 6;
		tyP0930MagConv1.tyFB.tyBtnRemoteUnclamp.usiTxtIdx:= 6;
	ELSE
		tyP0930MagConv1.tyFB.tyBtnFixedClamp.usiTxtIdx	:= 6;
		tyP0930MagConv1.tyFB.tyBtnFixedUnclamp.usiTxtIdx:= 6;
		tyP0930MagConv1.tyFB.tyBtnRemoteClamp.usiTxtIdx	:= 6;
		tyP0930MagConv1.tyFB.tyBtnRemoteUnclamp.usiTxtIdx:= 6;

	END_IF

	IF p_tyNtParamCurr.bMagAutoVerifyPrep = FALSE THEN
		IF tyP0930MagConv1.tyCom.tyBtnSwitch.bValue THEN
			fUIInRtStatHide(ADR(tyP0930MagConv1.tyFB.tyLyr.uiRtStat));
			fUIInRtStatHide(ADR(tyP0930MagConv1.tyDC.tyLyr.uiRtStat));
			fUIInRtStatHide(ADR(tyP0930MagConv1.tyFB.tyLyrWithoutSelClamp.uiRtStat));
			fUIInRtStatOff(ADR(tyP0930MagConv1.tyDC.tyLyrWithoutSelClamp.uiRtStat));
		ELSE
			fUIInRtStatHide(ADR(tyP0930MagConv1.tyFB.tyLyr.uiRtStat));
			fUIInRtStatHide(ADR(tyP0930MagConv1.tyDC.tyLyr.uiRtStat));
			fUIInRtStatOff(ADR(tyP0930MagConv1.tyFB.tyLyrWithoutSelClamp.uiRtStat));
			fUIInRtStatHide(ADR(tyP0930MagConv1.tyDC.tyLyrWithoutSelClamp.uiRtStat));
		END_IF
	ELSE
		IF tyP0930MagConv1.tyCom.tyBtnSwitch.bValue THEN
			fUIInRtStatHide(ADR(tyP0930MagConv1.tyFB.tyLyr.uiRtStat));
			fUIInRtStatOff(ADR(tyP0930MagConv1.tyDC.tyLyr.uiRtStat));
			fUIInRtStatHide(ADR(tyP0930MagConv1.tyFB.tyLyrWithoutSelClamp.uiRtStat));
			fUIInRtStatHide(ADR(tyP0930MagConv1.tyDC.tyLyrWithoutSelClamp.uiRtStat));
		ELSE
			fUIInRtStatOff(ADR(tyP0930MagConv1.tyFB.tyLyr.uiRtStat));
			fUIInRtStatHide(ADR(tyP0930MagConv1.tyDC.tyLyr.uiRtStat));
			fUIInRtStatHide(ADR(tyP0930MagConv1.tyFB.tyLyrWithoutSelClamp.uiRtStat));
			fUIInRtStatHide(ADR(tyP0930MagConv1.tyDC.tyLyrWithoutSelClamp.uiRtStat));
		END_IF
	END_IF

END_ACTION
```

#### Act_OptP0930FullMask.st
```iecst
ACTION Act_OptP0930FullMask:

	IF eCurrPage = UIP0930MagConv1 THEN

		IF p_tyDI.bEStopSig = FALSE THEN
			p_tyC0002FullMask ACCESS ADR(tyP0930MagConv1.tyFullMaskEStop);

		ELSIF p_tyDI.bCoverSWSig = FALSE THEN
			p_tyC0002FullMask ACCESS ADR(tyP0930MagConv1.tyFullMaskCWSig);

		ELSIF p_tyDI.bSafetyRlySig = FALSE THEN
			p_tyC0002FullMask ACCESS ADR(tyP0930MagConv1.tyFullMaskSafetyRly);

		ELSE
			p_tyC0002FullMask ACCESS ADR(tyP0930MagConv1.tyFullMaskHide);

		END_IF

	END_IF

END_ACTION
```

#### Act_OptP0930MagConv1ChgLyr.st
```iecst
ACTION Act_OptP0930MagConv1ChgLyr:

	IF p_tyNtParamCurr.bMagAutoVerifyPrep THEN
		IF tyP0930MagConv1.tyCom.tyBtnSwitch.bRtCompl THEN
			tyP0930MagConv1.tyCom.tyBtnSwitch.bRtCompl	:= FALSE;

			IF tyP0930MagConv1.tyCom.tyBtnSwitch.bValue = TRUE THEN
				fUIInRtStatOff(ADR(tyP0930MagConv1.tyDC.tyLyr.uiRtStat));
				fUIInRtStatHide(ADR(tyP0930MagConv1.tyFB.tyLyr.uiRtStat));
			ELSE
				fUIInRtStatHide(ADR(tyP0930MagConv1.tyDC.tyLyr.uiRtStat));
				fUIInRtStatOff(ADR(tyP0930MagConv1.tyFB.tyLyr.uiRtStat));
			END_IF

		END_IF
	ELSE
		IF tyP0930MagConv1.tyCom.tyBtnSwitch.bRtCompl THEN
			tyP0930MagConv1.tyCom.tyBtnSwitch.bRtCompl	:= FALSE;

			IF tyP0930MagConv1.tyCom.tyBtnSwitch.bValue = TRUE THEN
				fUIInRtStatOff(ADR(tyP0930MagConv1.tyDC.tyLyrWithoutSelClamp.uiRtStat));
				fUIInRtStatHide(ADR(tyP0930MagConv1.tyFB.tyLyrWithoutSelClamp.uiRtStat));
			ELSE
				fUIInRtStatHide(ADR(tyP0930MagConv1.tyDC.tyLyrWithoutSelClamp.uiRtStat));
				fUIInRtStatOff(ADR(tyP0930MagConv1.tyFB.tyLyrWithoutSelClamp.uiRtStat));
			END_IF

		END_IF
	END_IF

END_ACTION
```

#### Act_OptP0930MagConv1DC.st
```iecst
ACTION Act_OptP0930MagConv1DC:

	//Magazine Conveyor
	IF tyP0930MagConv1.tyDC.tyBtnStop.bRtCompl = TRUE THEN
		eMagConv2Clp1Act	:= MagConv2ClpActStop;

		IF p_eMagConv2Clp1Stat = MagConv2ClpActStop AND p_eMagConv2Clp1Status = Done THEN
			eMagConv2Clp1Act	:= MagConv2ClpActIdle;

			tyP0930MagConv1.tyDC.tyBtnStop.bRtCompl		:= FALSE;
			tyP0930MagConv1.tyDC.tyBtnStop.bValue		:= TRUE;
			tyP0930MagConv1.tyDC.tyBtnStop.bRtLk		:= TRUE;

			tyP0930MagConv1.tyDC.tyBtnMagIn.bRtCompl	:= FALSE;
			tyP0930MagConv1.tyDC.tyBtnMagIn.bValue		:= FALSE;
			tyP0930MagConv1.tyDC.tyBtnMagIn.bRtLk		:= FALSE;

			tyP0930MagConv1.tyDC.tyBtnMagOut.bRtCompl	:= FALSE;
			tyP0930MagConv1.tyDC.tyBtnMagOut.bValue		:= FALSE;
			tyP0930MagConv1.tyDC.tyBtnMagOut.bRtLk		:= FALSE;
		END_IF

	ELSIF tyP0930MagConv1.tyDC.tyBtnMagIn.bRtCompl = TRUE THEN
		tyP0930MagConv1.tyDC.tyBtnMagIn.bValue	:= TRUE;
		tyP0930MagConv1.tyDC.tyBtnMagIn.bRtLk	:= TRUE;

		tyP0930MagConv1.tyDC.tyBtnStop.bValue	:= FALSE;
		tyP0930MagConv1.tyDC.tyBtnStop.bRtLk	:= FALSE;

		IF p_tyNtParamCurr.eProjMagConvDir = ConvDirLToR OR p_tyNtParamCurr.eProjMagConvDir = ConvDirLToL THEN

			eMagConv2Clp1Act	:= MagConv2ClpActSetMtrSigOnOrLToR;

			IF p_eMagConv2Clp1Stat = MagConv2ClpActSetMtrSigOnOrLToR AND p_eMagConv2Clp1Status = Done THEN
				eMagConv2Clp1Act	:= MagConv2ClpActIdle;

				tyP0930MagConv1.tyDC.tyBtnMagIn.bRtCompl	:= FALSE;
			END_IF

		ELSE

			eMagConv2Clp1Act	:= MagConv2ClpActSetMtrDirOrRToL;

			IF p_eMagConv2Clp1Stat = MagConv2ClpActSetMtrDirOrRToL AND p_eMagConv2Clp1Status = Done THEN
				eMagConv2Clp1Act	:= MagConv2ClpActIdle;

				tyP0930MagConv1.tyDC.tyBtnMagIn.bRtCompl	:= FALSE;
			END_IF

		END_IF

	ELSIF tyP0930MagConv1.tyDC.tyBtnMagOut.bRtCompl = TRUE THEN
		tyP0930MagConv1.tyDC.tyBtnMagOut.bValue	:= TRUE;
		tyP0930MagConv1.tyDC.tyBtnMagOut.bRtLk	:= TRUE;

		tyP0930MagConv1.tyDC.tyBtnStop.bValue	:= FALSE;
		tyP0930MagConv1.tyDC.tyBtnStop.bRtLk	:= FALSE;

		IF p_tyNtParamCurr.eProjMagConvDir = ConvDirLToR OR p_tyNtParamCurr.eProjMagConvDir = ConvDirRToR THEN

			eMagConv2Clp1Act	:= MagConv2ClpActSetMtrSigOnOrLToR;

			IF p_eMagConv2Clp1Stat = MagConv2ClpActSetMtrSigOnOrLToR AND p_eMagConv2Clp1Status = Done THEN
				eMagConv2Clp1Act	:= MagConv2ClpActIdle;

				tyP0930MagConv1.tyDC.tyBtnMagOut.bRtCompl	:= FALSE;
			END_IF

		ELSE

			eMagConv2Clp1Act	:= MagConv2ClpActSetMtrDirOrRToL;

			IF p_eMagConv2Clp1Stat = MagConv2ClpActSetMtrDirOrRToL AND p_eMagConv2Clp1Status = Done THEN
				eMagConv2Clp1Act	:= MagConv2ClpActIdle;

				tyP0930MagConv1.tyDC.tyBtnMagOut.bRtCompl	:= FALSE;
			END_IF

		END_IF

	END_IF

	//Magazine Clamper
	IF tyP0930MagConv1.tyCom.tyBtnSwitch.bValue = TRUE THEN
		IF p_bSelClamp1TwoCtrlOut = FALSE THEN
			IF tyP0930MagConv1.tyDC.tyBtnSelUnclamp.bRtCompl = TRUE THEN
				tyP0930MagConv1.tyDC.tyBtnSelUnclamp.bValue := TRUE;
				tyP0930MagConv1.tyDC.tyBtnSelClamp.bValue := FALSE;

				eMagConvSelClp1Act	:= PneuActSetExt;

				IF p_eSelClamp1Stat = PneuActSetExt AND p_eSelClamp1Status = Done THEN
					eMagConvSelClp1Act	:= PneuActIdle;

					tyP0930MagConv1.tyDC.tyBtnSelUnclamp.bRtCompl	:= FALSE;
				END_IF

			ELSIF tyP0930MagConv1.tyDC.tyBtnSelClamp.bRtCompl = TRUE THEN
				tyP0930MagConv1.tyDC.tyBtnSelClamp.bValue := TRUE;
				tyP0930MagConv1.tyDC.tyBtnSelUnclamp.bValue := FALSE;

				eMagConvSelClp1Act	:= PneuActSetRet;

				IF p_eSelClamp1Stat = PneuActSetRet AND p_eSelClamp1Status = Done THEN
					eMagConvSelClp1Act	:= PneuActIdle;

					tyP0930MagConv1.tyDC.tyBtnSelClamp.bRtCompl	:= FALSE;
				END_IF
			END_IF

		ELSE
			IF (tyP0930MagConv1.tyDC.tyBtnSelUnclamp.bRtCompl = TRUE) OR (tyP0930MagConv1.tyDC.tyBtnSelClamp.bRtCompl = TRUE) THEN
				IF (tyP0930MagConv1.tyDC.tyBtnSelUnclamp.bValue = TRUE) AND (tyP0930MagConv1.tyDC.tyBtnSelClamp.bValue = TRUE) THEN
					eMagConvSelClp1Act	:= PneuActSetAll;

					IF p_eSelClamp1Stat = PneuActSetAll AND p_eSelClamp1Status = Done THEN
						eMagConvSelClp1Act	:= PneuActIdle;

						tyP0930MagConv1.tyDC.tyBtnSelUnclamp.bRtCompl		:= FALSE;
						tyP0930MagConv1.tyDC.tyBtnSelClamp.bRtCompl			:= FALSE;
					END_IF

				ELSIF (tyP0930MagConv1.tyDC.tyBtnSelUnclamp.bValue = TRUE) AND (tyP0930MagConv1.tyDC.tyBtnSelClamp.bValue = FALSE) THEN
					eMagConvSelClp1Act	:= PneuActSetRet;

					IF p_eSelClamp1Stat = PneuActSetRet AND p_eSelClamp1Status = Done THEN
						eMagConvSelClp1Act	:= PneuActIdle;

						tyP0930MagConv1.tyDC.tyBtnSelUnclamp.bRtCompl		:= FALSE;
						tyP0930MagConv1.tyDC.tyBtnSelClamp.bRtCompl			:= FALSE;
					END_IF

				ELSIF (tyP0930MagConv1.tyDC.tyBtnSelUnclamp.bValue = FALSE) AND (tyP0930MagConv1.tyDC.tyBtnSelClamp.bValue = TRUE) THEN
					eMagConvSelClp1Act	:= PneuActSetExt;

					IF p_eSelClamp1Stat = PneuActSetExt AND p_eSelClamp1Status = Done THEN
						eMagConvSelClp1Act	:= PneuActIdle;

						tyP0930MagConv1.tyDC.tyBtnSelUnclamp.bRtCompl		:= FALSE;
						tyP0930MagConv1.tyDC.tyBtnSelClamp.bRtCompl			:= FALSE;
					END_IF

				ELSE
					eMagConvSelClp1Act	:= PneuActRstAll;

					IF p_eSelClamp1Stat = PneuActRstAll AND p_eSelClamp1Status = Done THEN
						eMagConvSelClp1Act	:= PneuActIdle;

						tyP0930MagConv1.tyDC.tyBtnSelUnclamp.bRtCompl		:= FALSE;
						tyP0930MagConv1.tyDC.tyBtnSelClamp.bRtCompl			:= FALSE;
					END_IF

				END_IF
			END_IF
		END_IF

		IF p_bMagConv2Clp1ClprTwoOutputCtrl = FALSE THEN

			//Fixed
			IF tyP0930MagConv1.tyDC.tyBtnFixedClamp.bRtCompl = TRUE THEN
				tyP0930MagConv1.tyDC.tyBtnFixedClamp.bValue		:= TRUE;
				tyP0930MagConv1.tyDC.tyBtnFixedUnclamp.bValue	:= FALSE;

				eMagConv2Clp1Act	:= MagConv2ClpActFixClprSetClamp;

				IF p_eMagConv2Clp1Stat = MagConv2ClpActFixClprSetClamp AND p_eMagConv2Clp1Status = Done THEN
					eMagConv2Clp1Act	:= MagConv2ClpActIdle;

					tyP0930MagConv1.tyDC.tyBtnFixedClamp.bRtCompl	:= FALSE;
				END_IF

			ELSIF tyP0930MagConv1.tyDC.tyBtnFixedUnclamp.bRtCompl = TRUE THEN
				tyP0930MagConv1.tyDC.tyBtnFixedUnclamp.bValue	:= TRUE;
				tyP0930MagConv1.tyDC.tyBtnFixedClamp.bValue		:= FALSE;

				eMagConv2Clp1Act	:= MagConv2ClpActFixClprSetUnclamp;

				IF p_eMagConv2Clp1Stat = MagConv2ClpActFixClprSetUnclamp AND p_eMagConv2Clp1Status = Done THEN
					eMagConv2Clp1Act	:= MagConv2ClpActIdle;

					tyP0930MagConv1.tyDC.tyBtnFixedUnclamp.bRtCompl	:= FALSE;
				END_IF

			END_IF

			//Remote
			IF tyP0930MagConv1.tyDC.tyBtnRemoteClamp.bRtCompl = TRUE THEN
				tyP0930MagConv1.tyDC.tyBtnRemoteClamp.bValue		:= TRUE;
				tyP0930MagConv1.tyDC.tyBtnRemoteUnclamp.bValue		:= FALSE;

				eMagConv2Clp1Act	:= MagConv2ClpActRmtClprSetClamp;

				IF p_eMagConv2Clp1Stat = MagConv2ClpActRmtClprSetClamp AND p_eMagConv2Clp1Status = Done THEN
					eMagConv2Clp1Act	:= MagConv2ClpActIdle;

					tyP0930MagConv1.tyDC.tyBtnRemoteClamp.bRtCompl	:= FALSE;
				END_IF

			ELSIF tyP0930MagConv1.tyDC.tyBtnRemoteUnclamp.bRtCompl = TRUE THEN
				tyP0930MagConv1.tyDC.tyBtnRemoteUnclamp.bValue	:= TRUE;
				tyP0930MagConv1.tyDC.tyBtnRemoteClamp.bValue	:= FALSE;

				eMagConv2Clp1Act	:= MagConv2ClpActRmtClprSetUnclamp;

				IF p_eMagConv2Clp1Stat = MagConv2ClpActRmtClprSetUnclamp AND p_eMagConv2Clp1Status = Done THEN
					eMagConv2Clp1Act	:= MagConv2ClpActIdle;

					tyP0930MagConv1.tyDC.tyBtnRemoteUnclamp.bRtCompl	:= FALSE;
				END_IF

			END_IF

		ELSE

			//Fixed
			IF (tyP0930MagConv1.tyDC.tyBtnFixedClamp.bRtCompl = TRUE) OR (tyP0930MagConv1.tyDC.tyBtnFixedUnclamp.bRtCompl = TRUE) THEN

				IF (tyP0930MagConv1.tyDC.tyBtnFixedClamp.bValue = TRUE) AND (tyP0930MagConv1.tyDC.tyBtnFixedUnclamp.bValue = TRUE) THEN

					eMagConv2Clp1Act	:= MagConv2ClpActFixClprSetAll;

					IF p_eMagConv2Clp1Stat = MagConv2ClpActFixClprSetAll AND p_eMagConv2Clp1Status = Done THEN

						eMagConv2Clp1Act	:= MagConv2ClpActIdle;

						tyP0930MagConv1.tyDC.tyBtnFixedClamp.bRtCompl	:= FALSE;
						tyP0930MagConv1.tyDC.tyBtnFixedUnclamp.bRtCompl	:= FALSE;
					END_IF

				ELSIF (tyP0930MagConv1.tyDC.tyBtnFixedClamp.bValue = TRUE) AND (tyP0930MagConv1.tyDC.tyBtnFixedUnclamp.bValue = FALSE) THEN
					eMagConv2Clp1Act	:= MagConv2ClpActFixClprSetClamp;

					IF p_eMagConv2Clp1Stat = MagConv2ClpActFixClprSetClamp AND p_eMagConv2Clp1Status = Done THEN

						eMagConv2Clp1Act	:= MagConv2ClpActIdle;

						tyP0930MagConv1.tyDC.tyBtnFixedClamp.bRtCompl	:= FALSE;
						tyP0930MagConv1.tyDC.tyBtnFixedUnclamp.bRtCompl	:= FALSE;
					END_IF

				ELSIF (tyP0930MagConv1.tyDC.tyBtnFixedClamp.bValue = FALSE) AND (tyP0930MagConv1.tyDC.tyBtnFixedUnclamp.bValue = TRUE) THEN
					eMagConv2Clp1Act	:= MagConv2ClpActFixClprSetUnclamp;

					IF p_eMagConv2Clp1Stat = MagConv2ClpActFixClprSetUnclamp AND p_eMagConv2Clp1Status = Done THEN

						eMagConv2Clp1Act	:= MagConv2ClpActIdle;

						tyP0930MagConv1.tyDC.tyBtnFixedClamp.bRtCompl	:= FALSE;
						tyP0930MagConv1.tyDC.tyBtnFixedUnclamp.bRtCompl	:= FALSE;
					END_IF

				ELSE
					eMagConv2Clp1Act	:= MagConv2ClpActFixClprRstAll;

					IF p_eMagConv2Clp1Stat = MagConv2ClpActFixClprRstAll AND p_eMagConv2Clp1Status = Done THEN

						eMagConv2Clp1Act	:= MagConv2ClpActIdle;

						tyP0930MagConv1.tyDC.tyBtnFixedClamp.bRtCompl	:= FALSE;
						tyP0930MagConv1.tyDC.tyBtnFixedUnclamp.bRtCompl	:= FALSE;
					END_IF

				END_IF

				//Remote
				IF (tyP0930MagConv1.tyDC.tyBtnRemoteClamp.bRtCompl = TRUE) OR (tyP0930MagConv1.tyDC.tyBtnRemoteUnclamp.bRtCompl = TRUE) THEN

					IF (tyP0930MagConv1.tyDC.tyBtnRemoteClamp.bValue = TRUE) AND (tyP0930MagConv1.tyDC.tyBtnRemoteUnclamp.bValue = TRUE) THEN

						eMagConv2Clp1Act	:= MagConv2ClpActRmtClprSetAll;

						IF p_eMagConv2Clp1Stat = MagConv2ClpActRmtClprSetAll AND p_eMagConv2Clp1Status = Done THEN

							eMagConv2Clp1Act	:= MagConv2ClpActIdle;

							tyP0930MagConv1.tyDC.tyBtnRemoteClamp.bRtCompl		:= FALSE;
							tyP0930MagConv1.tyDC.tyBtnRemoteUnclamp.bRtCompl	:= FALSE;
						END_IF

					ELSIF (tyP0930MagConv1.tyDC.tyBtnRemoteClamp.bValue = TRUE) AND (tyP0930MagConv1.tyDC.tyBtnRemoteUnclamp.bValue = FALSE) THEN
						eMagConv2Clp1Act	:= MagConv2ClpActRmtClprSetClamp;

						IF p_eMagConv2Clp1Stat = MagConv2ClpActRmtClprSetClamp AND p_eMagConv2Clp1Status = Done THEN

							eMagConv2Clp1Act	:= MagConv2ClpActIdle;

							tyP0930MagConv1.tyDC.tyBtnRemoteClamp.bRtCompl	:= FALSE;
							tyP0930MagConv1.tyDC.tyBtnRemoteUnclamp.bRtCompl	:= FALSE;
						END_IF

					ELSIF (tyP0930MagConv1.tyDC.tyBtnRemoteClamp.bValue = FALSE) AND (tyP0930MagConv1.tyDC.tyBtnRemoteUnclamp.bValue = TRUE) THEN
						eMagConv2Clp1Act	:= MagConv2ClpActRmtClprSetUnclamp;

						IF p_eMagConv2Clp1Stat = MagConv2ClpActRmtClprSetUnclamp AND p_eMagConv2Clp1Status = Done THEN

							eMagConv2Clp1Act	:= MagConv2ClpActIdle;

							tyP0930MagConv1.tyDC.tyBtnRemoteClamp.bRtCompl	:= FALSE;
							tyP0930MagConv1.tyDC.tyBtnRemoteUnclamp.bRtCompl	:= FALSE;
						END_IF

					ELSE
						eMagConv2Clp1Act	:= MagConv2ClpActRmtClprRstAll;

						IF p_eMagConv2Clp1Stat = MagConv2ClpActRmtClprRstAll AND p_eMagConv2Clp1Status = Done THEN

							eMagConv2Clp1Act	:= MagConv2ClpActIdle;

							tyP0930MagConv1.tyDC.tyBtnRemoteClamp.bRtCompl	:= FALSE;
							tyP0930MagConv1.tyDC.tyBtnRemoteUnclamp.bRtCompl	:= FALSE;
						END_IF

					END_IF
				END_IF

			END_IF

		END_IF

		//Fixed
		tyP0930MagConv1.tyFB.tyBtnFixedClamp.bRtCompl		:= FALSE;
		tyP0930MagConv1.tyFB.tyBtnFixedClamp.bValue			:= FALSE;
		tyP0930MagConv1.tyFB.tyBtnFixedUnclamp.bRtCompl		:= FALSE;
		tyP0930MagConv1.tyFB.tyBtnFixedUnclamp.bValue		:= FALSE;

		//Remote
		tyP0930MagConv1.tyFB.tyBtnRemoteClamp.bRtCompl		:= FALSE;
		tyP0930MagConv1.tyFB.tyBtnRemoteClamp.bValue		:= FALSE;
		tyP0930MagConv1.tyFB.tyBtnRemoteUnclamp.bRtCompl	:= FALSE;
		tyP0930MagConv1.tyFB.tyBtnRemoteUnclamp.bValue		:= FALSE;

		//Top
		tyP0930MagConv1.tyFB.tyBtnSelClamp.bRtCompl		:= FALSE;
		tyP0930MagConv1.tyFB.tyBtnSelClamp.bValue		:= FALSE;
		tyP0930MagConv1.tyFB.tyBtnSelUnclamp.bRtCompl	:= FALSE;
		tyP0930MagConv1.tyFB.tyBtnSelUnclamp.bValue		:= FALSE;
	END_IF

	//Mask
	IF p_eMagConv2Clp1Status = Error THEN

		fUIInRtStatOff(ADR(tyP0930MagConv1.tyDC.tyBtnMagIn.uiMaskRtStat));
		fUIInRtStatOff(ADR(tyP0930MagConv1.tyDC.tyBtnMagOut.uiMaskRtStat));
		fUIInRtStatOff(ADR(tyP0930MagConv1.tyDC.tyBtnFixedClamp.uiMaskRtStat));
		fUIInRtStatOff(ADR(tyP0930MagConv1.tyDC.tyBtnFixedUnclamp.uiMaskRtStat));
		fUIInRtStatOff(ADR(tyP0930MagConv1.tyDC.tyBtnRemoteClamp.uiMaskRtStat));
		fUIInRtStatOff(ADR(tyP0930MagConv1.tyDC.tyBtnRemoteUnclamp.uiMaskRtStat));
		fUIInRtStatOff(ADR(tyP0930MagConv1.tyDC.tyBtnSelClamp.uiMaskRtStat));
		fUIInRtStatOff(ADR(tyP0930MagConv1.tyDC.tyBtnSelUnclamp.uiMaskRtStat));

	ELSIF tyP0930MagConv1.tyDC.tyBtnMagIn.bValue = TRUE THEN

		fUIInRtStatHide(ADR(tyP0930MagConv1.tyDC.tyBtnMagIn.uiMaskRtStat));
		fUIInRtStatOff(ADR(tyP0930MagConv1.tyDC.tyBtnMagOut.uiMaskRtStat));
		fUIInRtStatOff(ADR(tyP0930MagConv1.tyDC.tyBtnFixedClamp.uiMaskRtStat));
		fUIInRtStatOff(ADR(tyP0930MagConv1.tyDC.tyBtnFixedUnclamp.uiMaskRtStat));
		fUIInRtStatOff(ADR(tyP0930MagConv1.tyDC.tyBtnRemoteClamp.uiMaskRtStat));
		fUIInRtStatOff(ADR(tyP0930MagConv1.tyDC.tyBtnRemoteUnclamp.uiMaskRtStat));
		fUIInRtStatOff(ADR(tyP0930MagConv1.tyDC.tyBtnSelClamp.uiMaskRtStat));
		fUIInRtStatOff(ADR(tyP0930MagConv1.tyDC.tyBtnSelUnclamp.uiMaskRtStat));

	ELSIF tyP0930MagConv1.tyDC.tyBtnMagOut.bValue = TRUE THEN

		fUIInRtStatOff(ADR(tyP0930MagConv1.tyDC.tyBtnMagIn.uiMaskRtStat));
		fUIInRtStatHide(ADR(tyP0930MagConv1.tyDC.tyBtnMagOut.uiMaskRtStat));
		fUIInRtStatOff(ADR(tyP0930MagConv1.tyDC.tyBtnFixedClamp.uiMaskRtStat));
		fUIInRtStatOff(ADR(tyP0930MagConv1.tyDC.tyBtnFixedUnclamp.uiMaskRtStat));
		fUIInRtStatOff(ADR(tyP0930MagConv1.tyDC.tyBtnRemoteClamp.uiMaskRtStat));
		fUIInRtStatOff(ADR(tyP0930MagConv1.tyDC.tyBtnRemoteUnclamp.uiMaskRtStat));
		fUIInRtStatOff(ADR(tyP0930MagConv1.tyDC.tyBtnSelClamp.uiMaskRtStat));
		fUIInRtStatOff(ADR(tyP0930MagConv1.tyDC.tyBtnSelUnclamp.uiMaskRtStat));

	ELSE

		fUIInRtStatHide(ADR(tyP0930MagConv1.tyDC.tyBtnMagIn.uiMaskRtStat));
		fUIInRtStatHide(ADR(tyP0930MagConv1.tyDC.tyBtnMagOut.uiMaskRtStat));
		fUIInRtStatHide(ADR(tyP0930MagConv1.tyDC.tyBtnFixedClamp.uiMaskRtStat));
		fUIInRtStatHide(ADR(tyP0930MagConv1.tyDC.tyBtnFixedUnclamp.uiMaskRtStat));
		fUIInRtStatHide(ADR(tyP0930MagConv1.tyDC.tyBtnRemoteClamp.uiMaskRtStat));
		fUIInRtStatHide(ADR(tyP0930MagConv1.tyDC.tyBtnRemoteUnclamp.uiMaskRtStat));
		fUIInRtStatHide(ADR(tyP0930MagConv1.tyDC.tyBtnSelClamp.uiMaskRtStat));
		fUIInRtStatHide(ADR(tyP0930MagConv1.tyDC.tyBtnSelUnclamp.uiMaskRtStat));

	END_IF

END_ACTION
```
